Yaskawa INFORM job: SKRZYNIA_5540_-90_STOPNI_10BR.JBI

/JOB
//NAME SKRZYNIA_5540_-90_STOPNI_10BR
///FOLDERNAME 02-SKRZYNIE_JOBS
//POS
///NPOS 690,690,0,51,0,0
///TOOL 0
///POSTYPE PULSE
///PULSE
C00000=0,-52280,40443,0,6876,0
C00001=-82314,-24956,17040,-59626,-27382,-6248
C00002=-93910,-8625,17040,-59626,-43355,-6248
C00003=-98846,-1061,-42166,-80308,-57081,16120
C00004=-100452,6057,-48127,-85711,-56704,21322
C00005=-96957,25597,-37888,-85158,-62082,25522
C00006=-95580,33075,-33256,-84644,-64024,26851
C00007=-94380,33739,-32188,-85134,-63496,26721
C00008=-95580,33075,-33256,-84644,-64024,26851
C00009=-94940,31262,-36138,-85248,-63712,27160
C00010=-95580,33075,-33256,-84644,-64024,26851
C00011=-95263,33142,-33256,-84677,-63995,26850
C00012=-95263,33142,-33256,-84677,-63995,26850
C00013=-94261,33702,-32359,-85087,-63552,26740
C00014=-95263,33142,-33256,-84677,-63995,26850
C00015=-94777,31773,-35433,-85135,-63758,27084
C00016=-95263,33142,-33256,-84677,-63995,26850
C00017=-95260,33144,-33256,-84678,-63995,26850
C00018=-95260,33144,-33256,-84678,-63995,26850
C00019=-94282,33689,-32380,-85076,-63563,26742
C00020=-95260,33144,-33256,-84678,-63995,26850
C00021=-94827,31920,-35204,-85086,-63784,27059
C00022=-95260,33144,-33256,-84678,-63995,26850
C00023=-95258,33145,-33257,-84676,-63996,26846
C00024=-95258,33145,-33257,-84676,-63996,26846
C00025=-94286,33686,-32387,-85074,-63568,26738
C00026=-95258,33145,-33257,-84676,-63996,26846
C00027=-94874,32057,-34990,-85039,-63809,27032
C00028=-95258,33145,-33257,-84676,-63996,26846
C00029=-95258,33145,-33257,-84676,-63996,26846
C00030=-95258,33145,-33257,-84676,-63996,26846
C00031=-94323,33667,-32422,-85059,-63584,26741
C00032=-95258,33145,-33257,-84676,-63996,26846
C00033=-94899,32130,-34875,-85014,-63820,27019
C00034=-95258,33145,-33257,-84676,-63996,26846
C00035=-95258,25631,32269,-66559,-75499,2416
C00036=-95258,25631,32269,-66559,-75499,2416
C00037=-94333,26371,33350,-66433,-74983,2224
C00038=-95258,25631,32269,-66559,-75499,2416
C00039=-94886,24142,30119,-66602,-75133,2534
C00040=-95258,25631,32269,-66559,-75499,2416
C00041=-98646,19496,-17631,-99827,-80462,21224
C00042=-98811,21047,-15512,-99242,-81394,20987
C00043=-97886,21574,-14788,-99528,-80824,20997
C00044=-98811,21047,-15512,-99242,-81394,20987
C00045=-98517,19954,-17009,-99363,-81263,21101
C00046=-98811,21047,-15512,-99242,-81394,20987
C00047=-98811,19937,1242,-97498,-78933,15296
C00048=-98811,19937,1242,-97498,-78933,15296
C00049=-97933,20465,1962,-97646,-78345,15298
C00050=-98811,19937,1242,-97498,-78933,15296
C00051=-98523,18806,-285,-97586,-78782,15407
C00052=-98811,19937,1242,-97498,-78933,15296
C00053=-99152,37522,67957,-90787,-75030,-95
C00054=-99152,37522,67957,-90787,-75030,-95
C00055=-98279,38495,69612,-90504,-74443,-274
C00056=-99152,37522,67957,-90787,-75030,-95
C00057=-98708,34478,62881,-90983,-74820,488
C00058=-99152,37522,67957,-90787,-75030,-95
C00059=-98988,22776,44546,-90608,-68570,2568
C00060=-94428,854,16076,-89248,-50738,4740
C00061=-88080,-20128,-3199,-80943,-31244,2335
C00062=-50003,-39410,-5978,-16260,-18649,-25999
C00063=-48287,-44591,-17414,-16172,-14532,-25809
C00064=-91598,-4780,31748,-51735,-45731,-8771
C00065=-100979,4048,11685,-70926,-63965,7529
C00066=-99314,21122,10686,-75447,-74504,15845
C00067=-95042,27764,23446,-66422,-76166,12644
C00068=-94670,26279,21282,-66499,-75794,12766
C00069=-95042,27764,23446,-66422,-76166,12644
C00070=-94070,28550,24602,-66381,-75626,12438
C00071=-95042,27764,23446,-66422,-76166,12644
C00072=-97373,30352,38967,-71736,-79717,10385
C00073=-97373,30352,38967,-71736,-79717,10385
C00074=-96432,31128,40151,-71627,-79165,10198
C00075=-97373,30352,38967,-71736,-79717,10385
C00076=-97071,28917,36802,-71776,-79407,10544
C00077=-97373,30352,38967,-71736,-79717,10385
C00078=-97356,30262,38827,-71739,-79698,10398
C00079=-97356,30262,38827,-71739,-79698,10398
C00080=-96507,30957,39891,-71642,-79201,10230
C00081=-97356,30262,38827,-71739,-79698,10398
C00082=-97092,29010,36937,-71773,-79425,10538
C00083=-97356,30262,38827,-71739,-79698,10398
C00084=-97431,30641,39402,-71725,-79780,10352
C00085=-97431,30641,39402,-71725,-79780,10352
C00086=-96578,31348,40481,-71627,-79280,10181
C00087=-97431,30641,39402,-71725,-79780,10352
C00088=-97114,29116,37095,-71767,-79448,10523
C00089=-97431,30641,39402,-71725,-79780,10352
C00090=-99739,25677,21114,-82085,-78790,-4409
C00091=-99739,25677,21114,-82085,-78790,-4409
C00092=-98872,26250,21941,-82102,-78216,-4501
C00093=-99739,25677,21114,-82085,-78790,-4409
C00094=-99422,24232,19045,-82158,-78544,-4261
C00095=-99739,25677,21114,-82085,-78790,-4409
C00096=-98070,21699,18791,-100677,-76082,-5031
C00097=-98401,27942,27737,-100067,-79473,-6121
C00098=-97586,28537,28617,-100081,-78897,-6135
C00099=-98401,27942,27737,-100067,-79473,-6121
C00100=-98064,26400,25481,-100144,-79339,-5917
C00101=-98401,27942,27737,-100067,-79473,-6121
C00102=-99160,29228,35009,-99418,-79080,-8034
C00103=-98369,30564,38686,-99156,-78226,-8682
C00104=-97572,31199,39655,-99108,-77655,-8715
C00105=-98369,30564,38686,-99156,-78226,-8682
C00106=-98044,28949,36247,-99232,-78106,-8445
C00107=-98369,30564,38686,-99156,-78226,-8682
C00108=-99703,29561,37167,-99227,-79176,-8639
C00109=-98419,30528,38631,-99158,-78261,-8681
C00110=-98025,28599,35720,-99249,-78116,-8401
C00111=-98419,30528,38631,-99158,-78261,-8681
C00112=-97391,31350,39887,-99096,-77526,-8725
C00113=-98419,30528,38631,-99158,-78261,-8681
C00114=-91461,-8162,-10615,-106368,-48885,623
C00115=-98486,-14751,-40891,-114294,-59712,7739
C00116=-84089,-24462,-58822,-138905,-52068,17717
C00117=-93370,-29108,-64994,-133695,-56362,15444
C00118=-62749,-65297,-81682,-146767,-31843,20298
C00119=-73187,-23116,26488,-26118,-57509,-28469
C00120=-88600,6462,53521,-37454,-59134,-23478
C00121=-98388,13381,40686,-64111,-66922,-10378
C00122=-99819,33446,48735,-87787,-79679,-1235
C00123=-99819,33446,48735,-87787,-79679,-1235
C00124=-98945,34179,49898,-87659,-79086,-1350
C00125=-99819,33446,48735,-87787,-79679,-1235
C00126=-99591,32133,46677,-87830,-79529,-1033
C00127=-99819,33446,48735,-87787,-79679,-1235
C00128=-98853,28116,28355,-96898,-79749,4777
C00129=-98853,30464,37910,-96149,-78952,2546
C00130=-98284,30904,38579,-96116,-78548,2515
C00131=-98853,30464,37910,-96149,-78952,2546
C00132=-98656,29478,36421,-96191,-78865,2688
C00133=-98853,30464,37910,-96149,-78952,2546
C00134=-100018,29602,36606,-96210,-79777,2602
C00135=-100018,29602,36606,-96210,-79777,2602
C00136=-99324,30109,37370,-96174,-79287,2570
C00137=-99039,28675,35212,-96234,-79160,2773
C00138=-99324,30109,37370,-96174,-79287,2570
C00139=-98210,30963,38666,-96111,-78498,2511
C00140=-99324,30109,37370,-96174,-79287,2570
C00141=-94437,3365,15121,-90804,-55123,21
C00142=-76606,-19838,2636,-59027,-23020,-13375
C00143=-49667,-45532,-21960,-5654,-17518,-35856
C00144=-47485,-50287,-32535,-1070,-13732,-37871
///LIMIT ON
C00145=-36103,-65917,11738,-26975,4295,7905
///LIMIT OFF
C00146=-48283,-21883,28214,-25170,-26491,48363
C00147=-46664,-3144,58041,-18842,-32105,45325
C00148=-50347,-18571,12268,-49104,-16423,60029
C00149=-53571,-17125,12073,-56866,-17385,63433
C00150=-52069,-15730,13206,-55612,-16432,62999
C00151=-53474,-15384,13495,-57637,-17161,63825
C00152=-53571,-17125,12073,-56866,-17385,63433
C00153=-50509,-19000,10610,-51503,-15997,61182
C00154=-53130,-17211,12007,-56251,-17152,63186
C00155=-51822,-15992,12994,-55136,-16324,62798
C00156=-53635,-15431,13457,-57815,-17251,63894
C00157=-53130,-17211,12007,-56251,-17152,63186
C00158=-50704,-18403,11069,-52157,-16018,61478
C00159=-53231,-16470,14622,-53206,-17893,61673
C00160=-51756,-15101,15744,-51790,-16990,61165
C00161=-53741,-14453,16285,-54808,-17949,62397
C00162=-53231,-17580,11714,-56182,-17246,63139
C00163=-51814,-19410,10295,-53186,-16720,61844
C00164=-53629,-18979,7405,-62018,-16535,65958
C00165=-52238,-17698,8415,-61175,-15613,65699
C00166=-53551,-17401,8655,-62910,-16346,66402
C00167=-52880,-17654,11656,-55678,-17066,62935
C00168=-51005,-17995,11387,-52847,-16122,61778
C00169=-52964,-17611,11689,-55811,-17106,62990
C00170=-51611,-16353,12697,-54642,-16249,62582
C00171=-53495,-15765,13180,-57466,-17201,63739
C00172=-52964,-17611,11689,-55811,-17106,62990
C00173=-51030,-17982,11395,-52891,-16135,61798
C00174=-52975,-17563,11726,-55850,-17109,63009
C00175=-51607,-16289,12749,-54669,-16241,62596
C00176=-53283,-15811,13140,-57177,-17094,63622
C00177=-52975,-17563,11726,-55850,-17109,63009
C00178=-50945,-18019,11363,-52741,-16103,61737
C00179=-52728,-17788,11545,-55393,-17010,62816
C00180=-51045,-16207,12813,-53894,-15944,62287
C00181=-52895,-15647,13274,-56746,-16874,63461
C00182=-52728,-17788,11545,-55393,-17010,62816
C00183=-50945,-18019,11363,-52741,-16103,61737
C00184=-52556,-17520,11756,-55311,-16888,62798
C00185=-51113,-16157,12849,-54025,-15975,62343
C00186=-52730,-15718,13210,-56498,-16792,63358
C00187=-52556,-17520,11756,-55311,-16888,62798
C00188=-50945,-18019,11363,-52741,-16103,61737
C00189=-51893,-17787,11546,-54246,-16568,62356
C00190=-50379,-16341,12703,-52826,-15610,61849
C00191=-52406,-15704,13225,-56071,-16614,63190
C00192=-51893,-17787,11546,-54246,-16568,62356
C00193=-50028,-22953,-3957,-22347,-31919,54220
C00194=-50947,-22502,-3625,-23433,-32061,54736
C00195=-49421,-20951,-2455,-21951,-31329,54057
C00196=-51207,-20433,-2055,-24026,-31698,55041
C00197=-50529,-22709,-3778,-22940,-31995,54502
C00198=-49763,-25421,-36239,-24565,-26935,60445
C00199=-49763,-25421,-36239,-24565,-26935,60445
C00200=-48299,-23485,-34758,-23276,-26122,59713
C00201=-50218,-22723,-34165,-25568,-26529,60993
C00202=-49763,-25421,-36239,-24565,-26935,60445
C00203=-50713,-12366,-58367,-41124,-17813,74400
C00204=-50824,-12254,-58263,-41255,-17847,74484
C00205=-49431,-10052,-56192,-40383,-17131,73813
C00206=-50915,-9358,-55524,-41955,-17664,74847
C00207=-51028,-12852,-58814,-41301,-17980,74542
C00208=-49763,-25421,-36239,-24565,-26935,60445
C00209=-50529,-22709,-3778,-22940,-31995,54502
C00210=-45389,-28224,4312,-35967,-15579,54278
C00211=-40154,-51179,-915,-24203,-8234,36524
C00212=0,-52280,40443,0,6876,0
C00213=0,-52280,40443,0,6876,0
C00214=-2117,-50103,-33543,-4117,45077,85249
C00215=26439,-48928,-33543,-4117,-52362,85249
C00216=26439,-27355,-33543,-41485,-52362,85249
C00217=39218,-24492,-41653,-51934,-39374,86964
C00218=39218,-24492,-41653,-51934,-39374,86964
C00219=46639,7575,-9331,-26045,-41627,82486
C00220=47278,8641,-9483,-26175,-40625,82510
C00221=46369,10567,-7126,-26545,-41054,82831
C00222=47278,8641,-9483,-26175,-40625,82510
C00223=48256,9506,-8430,-25641,-40400,82076
C00224=47278,8641,-9483,-26175,-40625,82510
C00225=44522,-635,-31983,-49264,-28311,89687
C00226=44247,-628,-31975,-49394,-28443,89790
C00227=43310,1314,-29842,-49807,-28910,90140
C00228=44247,-628,-31975,-49394,-28443,89790
C00229=45313,152,-31124,-48894,-27920,89380
C00230=44247,-628,-31975,-49394,-28443,89790
C00231=41572,-13073,-22520,-50760,-38355,84033
C00232=21909,-6773,-14577,-94161,-56302,89381
C00233=23773,-3183,-10897,-94486,-55065,89563
C00234=24904,-823,-8382,-94654,-54308,89644
C00235=24395,1151,-6219,-94590,-54651,89617
C00236=24904,-823,-8382,-94654,-54308,89644
C00237=26178,-337,-7854,-94816,-53451,89710
C00238=24904,-823,-8382,-94654,-54308,89644
C00239=17020,-16061,-23281,-93084,-59494,88637
C00240=-21568,-26506,-31664,-90508,-85573,86639
C00241=-8557,-39769,-22319,-51419,-69406,84680
C00242=-8557,-39769,-22319,-51419,-69406,84680
C00243=32994,-9735,-10751,-29019,-59471,69498
C00244=43974,9628,-22604,-36190,-36396,73426
C00245=45932,13115,-22315,-37472,-33732,73846
C00246=45228,14664,-20329,-37571,-34159,74020
C00247=45932,13115,-22315,-37472,-33732,73846
C00248=46653,13731,-21526,-37109,-33514,73520
C00249=45932,13115,-22315,-37472,-33732,73846
C00250=39039,866,-6986,-42761,-44691,67687
C00251=30717,-9248,-22721,-77433,-42696,79486
C00252=32434,-7077,-20587,-77571,-41526,79457
C00253=31883,-5576,-19073,-77676,-41878,79560
C00254=32434,-7077,-20587,-77571,-41526,79457
C00255=33092,-6769,-20280,-77576,-41084,79417
C00256=32434,-7077,-20587,-77571,-41526,79457
C00257=30527,-14106,-27266,-76898,-42917,79150
C00258=25454,-9581,-17335,-94425,-53880,89429
C00259=24965,-2445,-10120,-94645,-54263,89631
C00260=24893,-1278,-8874,-94650,-54314,89639
C00261=24417,557,-6877,-94595,-54636,89618
C00262=24893,-1278,-8874,-94650,-54314,89639
C00263=25752,-956,-8526,-94759,-53737,89684
C00264=24893,-1278,-8874,-94650,-54314,89639
C00265=23817,-1527,-9142,-94518,-55040,89587
C00266=24871,-1152,-8735,-94651,-54328,89643
C00267=24440,508,-6926,-94601,-54619,89624
C00268=24871,-1152,-8735,-94651,-54328,89643
C00269=25635,-865,-8427,-94748,-53815,89684
C00270=24871,-1152,-8735,-94651,-54328,89643
C00271=33203,-4295,-13750,-123758,-49995,81034
C00272=35028,4195,-6818,-132965,-58836,87950
C00273=35028,4195,-6818,-132965,-58836,87950
C00274=34452,5837,-4911,-132720,-59045,87770
C00275=35028,4195,-6818,-132965,-58836,87950
C00276=35710,4593,-6360,-133217,-58512,88125
C00277=35028,4195,-6818,-132965,-58836,87950
C00278=24762,-11408,-28656,-113055,-60293,85383
C00279=-28645,-26349,-41223,-103369,-91870,78302
C00280=-28645,-26349,-41223,-103369,-91870,78302
C00281=-25549,-24286,-26215,-66769,-87032,80148
C00282=27561,-8271,-12315,-63268,-52553,74387
C00283=29336,-165,-3925,-63163,-51316,74265
C00284=29518,765,-2904,-63127,-51205,74233
C00285=28850,2962,-447,-63227,-51636,74327
C00286=29518,765,-2904,-63127,-51205,74233
C00287=30662,1292,-2320,-62902,-50501,74035
C00288=29518,765,-2904,-63127,-51205,74233
C00289=30773,10953,32136,-106912,-46141,83783
C00290=30773,10953,32136,-106912,-46141,83783
C00291=30080,13410,35293,-106601,-46463,83481
C00292=30773,10953,32136,-106912,-46141,83783
C00293=32007,11622,32987,-106899,-45346,83915
C00294=30773,10953,32136,-106912,-46141,83783
C00295=28321,-8642,-16372,-95739,-47180,89965
C00296=28583,-7344,-15096,-95864,-47019,90043
C00297=27897,-5229,-12965,-95873,-47499,90079
C00298=28583,-7344,-15096,-95864,-47019,90043
C00299=29900,-6813,-14567,-96101,-46141,90154
C00300=28583,-7344,-15096,-95864,-47019,90043
C00301=27852,-7537,-15286,-95742,-47508,89986
C00302=28448,-7306,-15058,-95845,-47110,90035
C00303=27795,-5283,-13021,-95851,-47567,90065
C00304=28448,-7306,-15058,-95845,-47110,90035
C00305=29772,-6774,-14527,-96083,-46226,90146
C00306=28448,-7306,-15058,-95845,-47110,90035
C00307=18552,-19531,-26179,-93438,-53589,88597
C00308=40301,-14999,-52277,-148979,-69262,86714
C00309=42323,-33,-37432,-150113,-69667,87489
C00310=53245,19091,3515,-165691,-72595,90030
C00311=53641,19552,4138,-165817,-72473,90151
C00312=53058,20743,5761,-165615,-72317,89948
C00313=53641,19552,4138,-165817,-72473,90151
C00314=54155,20160,4967,-165982,-72308,90306
C00315=53641,19552,4138,-165817,-72473,90151
C00316=23439,-10154,-17205,-109204,-58547,76547
C00317=2382,-21913,-40813,-107544,-74451,77239
C00318=-31257,-15877,-35733,-102288,-96107,74463
C00319=-39204,-18003,-7668,-86141,-99190,68413
C00320=-5592,-5690,18047,-75373,-79525,63129
C00321=19039,-439,25862,-68224,-64120,61443
C00322=21624,5223,26011,-69375,-61155,63193
C00323=24437,11840,34139,-68260,-59598,62567
C00324=24053,13588,36402,-68249,-59917,62491
C00325=24437,11840,34139,-68260,-59598,62567
C00326=25079,12112,34488,-68051,-59212,62472
C00327=24437,11840,34139,-68260,-59598,62567
C00328=21370,4935,25667,-69451,-61310,63230
C00329=-18351,-11002,3811,-80352,-86206,66275
C00330=-34619,-5846,8788,-82342,-97004,67025
C00331=-40684,-19963,-8478,-86482,-100204,67987
C00332=1570,-13136,-5998,-86227,-71173,69099
C00333=13966,-6596,-2340,-86587,-62612,70052
C00334=24093,-1862,-9504,-94546,-54850,89594
C00335=24093,-1862,-9504,-94546,-54850,89594
C00336=23519,425,-7024,-94488,-55240,89573
C00337=24093,-1862,-9504,-94546,-54850,89594
C00338=25256,-1442,-9053,-94693,-54067,89656
C00339=24093,-1862,-9504,-94546,-54850,89594
C00340=27718,4364,12871,-105518,-51077,86669
C00341=27718,4364,12871,-105518,-51077,86669
C00342=27164,6353,15202,-105385,-51398,86539
C00343=27718,4364,12871,-105518,-51077,86669
C00344=28828,4851,13441,-105618,-50355,86801
C00345=27718,4364,12871,-105518,-51077,86669
C00346=20930,-1364,27707,-95004,-52134,77785
C00347=-41463,-32191,18163,-91991,-64949,55938
C00348=0,-52277,40442,0,6872,4
C00349=-82314,-24956,17040,-59626,-27382,-6248
C00350=-93910,-8625,17040,-59626,-43355,-6248
C00351=-98846,-1061,-42166,-80308,-57081,16120
C00352=-100452,6057,-48127,-85711,-56704,21322
C00353=-95564,34698,-34234,-85516,-63941,27819
C00354=-94221,34299,-28769,-82558,-65564,25844
C00355=-94107,37241,-30442,-84005,-65307,27544
C00356=-95103,32620,-31323,-83378,-64939,26072
C00357=-95103,32620,-31323,-83378,-64939,26072
C00358=-93990,32828,-31380,-83932,-64473,26160
C00359=-94063,31710,-30585,-83283,-64598,25457
C00360=-96692,32939,-31211,-82617,-65723,26190
C00361=-96111,21840,170,-71736,-70232,11396
C00362=-94229,22391,773,-71789,-70557,11468
C00363=-94283,22521,1025,-71678,-70686,11433
C00364=-95675,19167,-4176,-72970,-68231,11735
C00365=-95681,24338,3488,-71459,-71669,11415
C00366=-94245,22750,1246,-71757,-70674,11453
C00367=-94341,22923,1499,-71729,-70746,11440
C00368=-96213,24222,3324,-71394,-71999,11479
C00369=-95517,23330,2066,-71543,-71508,11507
C00370=-94304,22892,1449,-71738,-70721,11443
C00371=-94158,22889,1452,-71756,-70627,11429
C00372=-96071,24319,3461,-71408,-71916,11455
C00373=-96941,-6406,-33809,-76117,-54125,10511
C00374=-89093,-33107,-44597,-67545,-52550,2722
C00375=-66103,-61757,7450,-21008,-32955,-5749
C00376=4223,-52290,40457,-5766,6913,3980
C00377=4223,-52290,40457,-5766,6913,3980
C00378=-4538,-50065,-33535,-3011,44998,84219
C00379=24207,-49248,-33668,-5551,-52644,86091
C00380=25094,-27722,-33812,-41887,-53054,85599
C00381=38036,-25052,-42086,-52219,-40087,87228
C00382=37328,-2824,-24733,-57182,-37821,90318
C00383=36700,-2520,-13735,-51589,-42201,86442
C00384=37520,2330,-3498,-48550,-43875,84431
C00385=37520,1020,-12079,-52650,-40851,87066
C00386=48458,-261,-12985,-24069,-43340,80504
C00387=36153,7296,-1758,-40139,-50302,89334
C00388=37146,11264,2520,-40849,-50296,89553
C00389=38059,11410,-1863,-40565,-47910,90206
C00390=36726,6476,-7858,-41213,-48206,90783
C00391=19339,7883,9818,-77509,-64249,74140
C00392=19027,1888,-16187,-103553,-67480,82955
C00393=24158,3537,-14322,-106039,-60939,84018
C00394=24143,4321,-7309,-103852,-59670,81875
C00395=19531,2904,-8928,-102027,-65985,80961
C00396=20232,-3383,-14682,-86495,-63009,78978
C00397=-24375,-51634,-49601,-83793,-94064,73950
C00398=4223,-52290,40457,-5766,6913,3980
C00399=-4825,-36686,24602,37792,-30278,35378
C00400=-46221,-29633,7403,-27051,-24124,46751
C00401=-46221,-29633,7403,-27051,-24124,46751
C00402=-52474,-20611,11454,-41004,-23045,52959
C00403=-60257,-19980,-2088,-84190,-23320,82051
C00404=-63868,-19883,-6318,-95759,-28031,88346
C00405=-51819,-22965,8574,-41365,-22900,53139
C00406=-4825,-36686,24602,37792,-30278,35378
C00407=-66103,-61757,7450,-21008,-32955,-5749
C00408=-89093,-33107,-44597,-67545,-52550,2722
C00409=-96941,-6406,-33809,-76117,-54125,10511
C00410=-99429,14378,84,-80785,-71596,8628
C00411=-99699,24313,24829,-82602,-77917,4569
C00412=-98066,26841,20697,-83331,-79245,6860
C00413=-98079,26929,20513,-83349,-79351,6953
C00414=-99638,19663,10292,-84193,-74452,7551
C00415=-99636,19665,10291,-84197,-74448,7550
C00416=-98131,26698,20177,-83371,-79212,6975
C00417=-98097,25980,12653,-84102,-79057,9159
C00418=-99636,19665,10291,-84197,-74448,7550
C00419=-99636,19665,10291,-84197,-74448,7550
C00420=-98186,26934,20517,-83350,-79332,6954
C00421=-98240,27087,20738,-83333,-79465,6940
C00422=-99636,19665,10291,-84197,-74448,7550
C00423=-99215,3992,8526,-80547,-63068,1835
C00424=-100264,1107,23397,-72827,-59854,-5092
C00425=-100264,1107,23397,-72827,-59854,-5092
C00426=-99514,-9483,18258,-71284,-60958,-4118
C00427=-61441,-38616,11032,-55510,-42874,-3049
C00428=4223,-52290,40457,-5766,6913,3980
C00429=-22331,-23394,-30093,-82917,-82006,85712
C00430=22434,-14401,-3235,-51104,-60845,74728
C00431=42744,21307,45077,-24753,-69813,65333
C00432=33655,14083,18147,-45417,-58301,71861
C00433=33641,11943,8279,-47835,-54840,73983
C00434=36574,13250,23432,-35354,-61822,69159
C00435=28497,326,20939,-70981,-47632,72427
C00436=30972,5983,29862,-68494,-46670,70994
C00437=31029,11571,45127,-63398,-49004,67378
C00438=28971,8096,39948,-65070,-49810,68216
C00439=29759,-12862,-24221,-91747,-41905,86600
C00440=35278,-10419,-21940,-93284,-36771,87139
C00441=36208,-10883,-22374,-93618,-35345,87231
C00442=27219,-23595,-33313,-89555,-43517,85303
C00443=10564,-40773,-45889,-85382,-54876,82708
C00444=-14984,-61618,-24572,-87392,-53367,60735
C00445=9346,-67436,-18786,-75708,-34590,53709
C00446=40938,-55232,35946,-9746,5421,6718
C00447=4223,-52290,40457,-5766,6913,3980
C00448=-4825,-36686,24602,37792,-30278,35378
C00449=-46221,-29633,7403,-27051,-24124,46751
C00450=-56796,-22932,368,-68953,-21567,70907
C00451=-61611,-20349,-6598,-95791,-25091,88405
C00452=-63740,-19715,-7390,-98604,-28245,90373
C00453=-52085,-22687,8760,-40927,-22666,52970
C00454=-49294,-34086,9663,-30689,-30758,52546
C00455=4223,-52290,40457,-5766,6913,3980
C00456=0,-52280,40443,0,6876,0
C00457=0,-52280,40443,0,6876,0
C00458=-61754,-61602,7279,-16215,-32140,-7126
C00459=-89313,-24027,20291,-53466,-58905,-4975
C00460=-97807,-25409,-21837,-78881,-62828,2121
C00461=-95644,-21015,-18476,-76474,-46020,1039
C00462=-99784,20282,11129,-84157,-74554,7499
C00463=-100058,25789,39872,-88643,-74345,1113
C00464=-98402,30585,40634,-89771,-78826,2411
C00465=-98157,28480,31016,-94616,-79375,5454
C00466=-99711,20530,18234,-96341,-74733,7105
C00467=-98387,24449,13333,-103557,-81562,10447
C00468=-96604,24297,13119,-103804,-80422,10626
C00469=-96604,26005,23528,-102938,-78741,7977
C00470=-99312,16704,-2418,-105415,-78692,13344
C00471=-99082,-15666,-17237,-92076,-50940,5911
C00472=-62624,-50447,-44776,-76934,-16957,-1114
C00473=-75165,-16680,32803,-38944,-52307,-27215
C00474=-75165,-16680,32803,-38944,-52307,-27215
C00475=-95350,8536,58133,-52477,-59539,-22352
C00476=-100948,11380,23586,-76731,-68346,-5781
C00477=-95677,27971,29253,-68711,-77159,-3356
C00478=-95583,25946,19380,-69779,-75412,-992
C00479=-98294,19288,21509,-68095,-73058,-4657
C00480=-100497,3428,15340,-68921,-63273,-8271
C00481=-81087,-35886,-14825,-53529,-36311,-18004
C00482=-47029,-49867,-20464,-11808,-29290,-36568
///LIMIT ON
C00483=-41431,-67449,10869,-1325,127,-6150
///LIMIT OFF
C00484=6328,-52297,40483,-8599,6957,5944
C00485=-8648,-69005,-18270,-84275,-43232,53472
C00486=18757,-59462,-34892,-84638,-37529,67311
C00487=26772,-23733,-33422,-89486,-43820,85275
C00488=29039,-10071,-21608,-91386,-45181,86629
C00489=29639,-5923,-17523,-91591,-45648,86808
C00490=29709,-5453,-17046,-91618,-45636,86826
C00491=29138,-10182,-21714,-91372,-45196,86624
C00492=20424,-22725,-32635,-88800,-51006,85261
C00493=28416,-11420,-25238,-98178,-46636,84572
C00494=30481,-6584,-16425,-92636,-44382,82541
C00495=30464,-7521,-23523,-96665,-44944,85234
C00496=28416,-11420,-25238,-98178,-46636,84572
C00497=-23524,-33387,-42654,-89891,-81168,80229
C00498=-23524,-33387,-42654,-89891,-81168,80229
C00499=33935,-6399,-10013,-60506,-43064,77980
C00500=34878,-3211,-6740,-60356,-42422,77865
C00501=34873,-3218,-6748,-60357,-42424,77868
C00502=33935,-6399,-10013,-60506,-43064,77980
C00503=17782,-19597,1250,-60925,-51448,69151
C00504=-243,-43047,-13224,-69794,-55957,65877
C00505=42700,-55269,36176,-13619,5333,9062
C00506=6328,-52297,40483,-8599,6957,5944
C00507=-10231,-60460,6271,71658,-11927,-13637
C00508=-49129,-39322,3023,-34904,-18609,43900
C00509=-57258,-19535,13114,-46502,-25798,55150
C00510=-58736,-19151,1344,-78268,-22199,76919
C00511=-56868,-17231,8572,-62431,-21728,66645
C00512=-56011,-29317,6725,-41009,-27363,52457
C00513=-10137,-60963,4526,62308,-14518,-6745
C00514=0,-52280,40443,0,6876,0
C00515=0,-52280,40443,0,6876,0
C00516=-41653,-63035,2931,-3578,-7576,-14589
C00517=-45770,-50109,-20524,-10089,-29273,-37310
C00518=-80544,-36303,-15042,-52975,-36116,-18265
C00519=-98926,-23964,-13239,-67549,-54178,-9552
C00520=-98901,-11554,-2908,-69008,-53412,-8360
C00521=-101174,454,-4800,-81790,-63681,-152
C00522=-100336,15373,10036,-81991,-73209,850
C00523=-98655,27908,24922,-81730,-79774,792
C00524=-98593,28720,26118,-81685,-80145,709
C00525=-99951,24070,19376,-82000,-77829,1145
C00526=-99951,24070,19376,-82000,-77829,1145
C00527=-98577,27118,23759,-81796,-79157,859
C00528=-98518,28577,26461,-81649,-79882,537
C00529=-99951,24070,19376,-82000,-77829,1145
C00530=-99951,24070,19376,-82000,-77829,1145
C00531=-98479,26563,22955,-81844,-78651,906
C00532=-98651,28095,26058,-81646,-79654,489
C00533=-99951,24070,19376,-82000,-77829,1145
C00534=-97595,-1409,-12320,-84284,-60474,1798
C00535=-100010,-16422,-27011,-84227,-53565,945
C00536=-88098,-29848,-22776,-71580,-48483,-7812
C00537=-81694,-37220,-20464,-64791,-45723,-12569
C00538=-45770,-50109,-20524,-10089,-29273,-37310
///LIMIT ON
C00539=-40984,-65135,6743,-2520,-4051,-10897
///LIMIT OFF
C00540=0,-52280,40443,0,6876,0
C00541=40939,-55232,35946,-9746,5421,6719
C00542=8707,-69002,-18268,-75213,-34271,52581
C00543=23267,-58917,-25142,-81990,-31707,62852
C00544=27307,-5613,10331,-81857,-46454,76095
C00545=30064,-5598,-963,-91827,-44222,81590
C00546=30419,-1725,5291,-88668,-43977,80354
C00547=30554,-300,10432,-88528,-43656,79164
C00548=29815,-6351,-3652,-90193,-44535,81892
C00549=29567,1847,27834,-65726,-48411,69959
C00550=23257,11670,30420,-81328,-57342,77033
C00551=23257,16856,45442,-77525,-58254,73578
C00552=21577,7912,33836,-78698,-59121,74340
C00553=17856,-9033,24892,-70658,-55966,67475
C00554=20838,-7097,2019,-111788,-62648,79114
C00555=40635,280,-7982,-142398,-56681,90238
C00556=32653,-9455,434,-90251,-40347,77213
C00557=40635,572,-6271,-142064,-55879,89947
C00558=40665,7761,2001,-141975,-55632,89869
C00559=40707,9678,10648,-140211,-51894,88431
C00560=39416,1907,3178,-139370,-51839,87774
C00561=7767,-21333,-19174,-120411,-69473,77116
C00562=33666,-18553,20064,-54519,-41956,59729
C00563=4032,-43511,13506,-33366,-30942,40837
C00564=22997,-56875,21315,16958,-8102,3163
C00565=0,-52280,40443,0,6876,0
///LIMIT ON
C00566=-50974,-46557,23391,-77768,-13896,42026
///LIMIT OFF
C00567=-53474,-39983,4253,-39182,-18848,44272
C00568=-56619,-19856,12878,-45665,-25558,54806
C00569=-53298,-26712,-11188,-26889,-32979,52528
C00570=-57200,-20845,-7559,-37425,-33513,53351
C00571=-58648,-23818,-25853,-45100,-31207,62168
C00572=-58477,-22145,-38977,-48305,-29254,64725
C00573=-51868,-27423,-11673,-25269,-32728,51737
C00574=-49121,-45409,-2608,-26656,-19965,38583
C00575=-21301,-61008,4568,43957,-10534,-712
C00576=0,-52280,40443,0,6876,0
C00577=0,-52280,40443,0,6876,0
///LIMIT ON
C00578=-40221,-67507,11044,-1325,-65,-6716
///LIMIT OFF
C00579=-45770,-50109,-20525,-10088,-29274,-37311
C00580=-80544,-36303,-15042,-52975,-36116,-18265
C00581=-97467,-10562,-5788,-76786,-47590,-5366
C00582=-98581,16268,9073,-102291,-74115,5399
C00583=-96245,23653,15791,-106069,-78604,6508
C00584=-96042,26225,19489,-105739,-79656,6032
C00585=-98519,17635,7561,-106659,-77043,7343
C00586=-98519,17635,7561,-106659,-77043,7343
C00587=-96298,25666,18652,-105800,-79560,6117
C00588=-95268,26547,15396,-109206,-81354,7908
C00589=-98519,17635,7561,-106659,-77043,7343
C00590=-98519,17635,7561,-106659,-77043,7343
C00591=-96096,27437,22144,-104884,-80110,5412
C00592=-96096,29559,32298,-104067,-78465,2996
C00593=-99245,17823,12181,-105373,-75632,5896
C00594=-101192,5225,-3909,-107580,-71003,7673
C00595=-100287,-3253,-24038,-111364,-68562,12025
C00596=-99412,-19117,-26908,-100833,-57247,5735
C00597=-91712,-30589,-22890,-72058,-50969,-7685
C00598=-81694,-37221,-20464,-64791,-45723,-12569
C00599=-45770,-50109,-20525,-10088,-29274,-37311
///LIMIT ON
C00600=-40221,-67507,11044,-1325,-65,-6716
///LIMIT OFF
C00601=0,-52280,40443,0,6876,0
C00602=51241,-30653,28678,4016,-29070,6398
C00603=46185,-61941,-37286,-12736,-10732,51851
C00604=-13205,-44768,-23966,-65315,-59418,73750
C00605=-11120,-40541,-20876,-69249,-61539,75403
C00606=-836,-13033,12361,-83908,-73576,73378
C00607=18912,6214,32354,-79489,-60743,73080
C00608=21217,10898,38129,-78632,-59343,72736
C00609=23447,16313,45262,-77527,-58074,72177
C00610=23610,23756,64158,-73325,-59549,68283
C00611=18912,6214,32354,-79489,-60743,73080
C00612=-836,-13033,12361,-83908,-73576,73378
C00613=-20209,-39682,-20467,-71924,-67122,76479
C00614=-20209,-39682,-20467,-71924,-67122,76479
C00615=26353,-3691,11741,-61723,-54035,71160
C00616=29598,-2090,11073,-69087,-47235,76987
C00617=30217,-1844,4641,-75777,-45517,79979
C00618=29529,1742,11379,-68166,-49318,73572
C00619=24010,-9039,-4437,-79986,-50972,77255
C00620=24652,-10740,-12845,-99298,-50700,81949
C00621=28976,-2672,-4778,-100308,-47937,82653
C00622=31030,-2921,-9996,-112394,-49006,86348
C00623=24652,-10740,-12845,-99298,-50700,81949
C00624=-25637,-26222,-38592,-96633,-85474,81576
C00625=-36771,-16470,-4689,-95304,-89579,74076
C00626=-33704,-12343,7746,-85568,-87064,70052
C00627=4032,-43511,13506,-33366,-30942,40837
C00628=27500,-60047,23168,28912,-2679,-5784
C00629=0,-52280,40443,0,6876,0
///LIMIT ON
C00630=-50971,-46557,23390,-77766,-13895,42026
///LIMIT OFF
C00631=-53475,-39984,4253,-39182,-18848,44273
C00632=-56619,-19856,12878,-45665,-25558,54806
C00633=-57643,-27958,-8553,-51854,-24771,59787
C00634=-66195,-24410,-19095,-90567,-31132,85904
C00635=-63290,-24193,-14362,-80030,-27547,78073
C00636=-39040,-40975,-15408,-18643,-21575,44866
C00637=-11647,-69843,-10959,56399,-11165,-4616
C00638=-15394,-57237,30542,-10392,5525,8219
C00639=0,-52280,40443,0,6876,0
C00640=0,-52280,40443,0,6876,0
///LIMIT ON
C00641=-40221,-67507,11044,-1325,-65,-6716
///LIMIT OFF
C00642=-45770,-50109,-20525,-10088,-29274,-37311
C00643=-94648,-18162,1575,-63292,-43035,-13570
C00644=-99112,3606,8889,-81344,-61742,-3619
C00645=-98572,26113,23382,-85571,-78492,509
C00646=-98656,28006,28806,-88976,-79248,97
C00647=-99839,24479,25828,-85077,-77001,-891
C00648=-99133,24879,24637,-94741,-77121,-2989
C00649=-98191,27052,27787,-94567,-78528,-3332
C00650=-98227,29022,36334,-93788,-77894,-5388
C00651=-100426,22466,21877,-95586,-77332,-2808
C00652=-99354,26201,32225,-100574,-76808,-3840
C00653=-96710,26250,34212,-100282,-74747,-4257
C00654=-96874,35880,54576,-99674,-76365,-9625
C00655=-99006,18159,13355,-102982,-74997,-2069
C00656=-97772,10218,8448,-107701,-67594,4685
C00657=-93425,-10069,4368,-74507,-47150,-8636
C00658=-96059,-18596,-7139,-76413,-48563,-7500
C00659=-96347,-8336,27647,-69083,-51241,-16001
C00660=-70313,-35289,-4922,-51188,-38634,-20596
C00661=-81694,-37221,-20464,-64791,-45723,-12569
C00662=-45770,-50109,-20525,-10088,-29274,-37311
C00663=-41628,-63095,3038,-3547,-7472,-14475
C00664=4223,-52290,40457,-5766,6913,3980
C00665=4224,-52288,40457,-5773,6909,3978
C00666=4224,-52288,40457,-28770,-64753,45638
C00667=6548,2882,44080,-77825,-67624,70557
C00668=22702,21750,69443,-66118,-61597,67582
C00669=25585,21999,63350,-62249,-61285,68688
C00670=25777,17209,50811,-62979,-59886,70957
C00671=23226,22825,71113,-65575,-61542,67353
C00672=24931,14697,51677,-80718,-51653,72069
C00673=24746,14409,39758,-87518,-53542,76879
C00674=24784,21556,58944,-82031,-53873,72431
C00675=22657,12722,42993,-85587,-54940,74916
C00676=-4427,-20395,-7318,-104668,-69521,79317
C00677=768,-20151,-3587,-97758,-65802,76626
C00678=-14736,-21545,-1233,-93598,-60476,72578
C00679=1642,-46684,14475,-47609,-24983,34912
C00680=27500,-60047,23168,28912,-2679,-5784
C00681=0,-52280,40443,0,6876,0
///LIMIT ON
C00682=-50971,-46557,23390,-77766,-13895,42026
///LIMIT OFF
C00683=-53475,-39984,4253,-39182,-18848,44273
C00684=-56619,-19856,12878,-45665,-25558,54806
C00685=-53891,-17708,14512,-43170,-23995,53902
C00686=-60674,-17500,6427,-71116,-24772,71097
C00687=-63181,-17997,2063,-82122,-26831,78394
C00688=-39402,-27697,7664,-17904,-21663,43170
C00689=-11647,-69843,-10959,56399,-11165,-4616
BC00000=479725
BC00001=460491
BC00002=460491
BC00003=460491
BC00004=460491
BC00005=460491
BC00006=460491
BC00007=460491
BC00008=460491
BC00009=460491
BC00010=460491
BC00011=506593
BC00012=506593
BC00013=506593
BC00014=506593
BC00015=506593
BC00016=506593
BC00017=552803
BC00018=552803
BC00019=552803
BC00020=552803
BC00021=552803
BC00022=552803
BC00023=598907
BC00024=598907
BC00025=598907
BC00026=598907
BC00027=598907
BC00028=598907
BC00029=621955
BC00030=621955
BC00031=621955
BC00032=621955
BC00033=621955
BC00034=621955
BC00035=574754
BC00036=574754
BC00037=574754
BC00038=574754
BC00039=574754
BC00040=574754
BC00041=620864
BC00042=620864
BC00043=620865
BC00044=620864
BC00045=620864
BC00046=620864
BC00047=620864
BC00048=620864
BC00049=620864
BC00050=620864
BC00051=620864
BC00052=620864
BC00053=619616
BC00054=619616
BC00055=619616
BC00056=619616
BC00057=619616
BC00058=619616
BC00059=619616
BC00060=619616
BC00061=619616
BC00062=619616
BC00063=714482
BC00064=722304
BC00065=754708
BC00066=767117
BC00067=767117
BC00068=767117
BC00069=767117
BC00070=767117
BC00071=767117
BC00072=752564
BC00073=752564
BC00074=752564
BC00075=752564
BC00076=752564
BC00077=752564
BC00078=798636
BC00079=798636
BC00080=798636
BC00081=798636
BC00082=798636
BC00083=798636
BC00084=821725
BC00085=821725
BC00086=821725
BC00087=821725
BC00088=821725
BC00089=821725
BC00090=858551
BC00091=858551
BC00092=858551
BC00093=858551
BC00094=858551
BC00095=858551
BC00096=864565
BC00097=864565
BC00098=864565
BC00099=864565
BC00100=864565
BC00101=864565
BC00102=879162
BC00103=879162
BC00104=879162
BC00105=879162
BC00106=879162
BC00107=879162
BC00108=916154
BC00109=916154
BC00110=916154
BC00111=916154
BC00112=916154
BC00113=916154
BC00114=887605
BC00115=887605
BC00116=887605
BC00117=887605
BC00118=887605
BC00119=974304
BC00120=974304
BC00121=984323
BC00122=988419
BC00123=988419
BC00124=988419
BC00125=988419
BC00126=988419
BC00127=988419
BC00128=1003836
BC00129=1003836
BC00130=1003836
BC00131=1003836
BC00132=1003836
BC00133=1003836
BC00134=1003836
BC00135=1048824
BC00136=1048824
BC00137=1048824
BC00138=1048824
BC00139=1048824
BC00140=1048824
BC00141=992185
BC00142=986127
BC00143=1002338
BC00144=951360
BC00145=873120
BC00146=935062
BC00147=935062
BC00148=964364
BC00149=966461
BC00150=966461
BC00151=966461
BC00152=966461
BC00153=904985
BC00154=904985
BC00155=904985
BC00156=904985
BC00157=904985
BC00158=843543
BC00159=843543
BC00160=843543
BC00161=843543
BC00162=843543
BC00163=782113
BC00164=782113
BC00165=782113
BC00166=782113
BC00167=782113
BC00168=720711
BC00169=720711
BC00170=720711
BC00171=720711
BC00172=720711
BC00173=659226
BC00174=659226
BC00175=659226
BC00176=659226
BC00177=659226
BC00178=597825
BC00179=597825
BC00180=597825
BC00181=597825
BC00182=597825
BC00183=536353
BC00184=536353
BC00185=536353
BC00186=536353
BC00187=536353
BC00188=474901
BC00189=474901
BC00190=474901
BC00191=474901
BC00192=474901
BC00193=474905
BC00194=474905
BC00195=474905
BC00196=474905
BC00197=474905
BC00198=474905
BC00199=474905
BC00200=474905
BC00201=474905
BC00202=474905
BC00203=474905
BC00204=474905
BC00205=474905
BC00206=474905
BC00207=474905
BC00208=474905
BC00209=474905
BC00210=474901
BC00211=548577
BC00212=548577
BC00213=492150
BC00214=423885
BC00215=423885
BC00216=423885
BC00217=423885
BC00218=423885
BC00219=493160
BC00220=493160
BC00221=493160
BC00222=493160
BC00223=493160
BC00224=493160
BC00225=539180
BC00226=539180
BC00227=539180
BC00228=539180
BC00229=539180
BC00230=539180
BC00231=525487
BC00232=485388
BC00233=485386
BC00234=485384
BC00235=485384
BC00236=485384
BC00237=485384
BC00238=485384
BC00239=485384
BC00240=485384
BC00241=485384
BC00242=635507
BC00243=635507
BC00244=635507
BC00245=635509
BC00246=635509
BC00247=635509
BC00248=635509
BC00249=635509
BC00250=603035
BC00251=594948
BC00252=594948
BC00253=594948
BC00254=594948
BC00255=594948
BC00256=594948
BC00257=594948
BC00258=600591
BC00259=600589
BC00260=600589
BC00261=600589
BC00262=600589
BC00263=600589
BC00264=600589
BC00265=623637
BC00266=623637
BC00267=623637
BC00268=623637
BC00269=623637
BC00270=623637
BC00271=623637
BC00272=623637
BC00273=623637
BC00274=623637
BC00275=623637
BC00276=623637
BC00277=623637
BC00278=623637
BC00279=623637
BC00280=758391
BC00281=758391
BC00282=758391
BC00283=758391
BC00284=758391
BC00285=758391
BC00286=758391
BC00287=758391
BC00288=758391
BC00289=669704
BC00290=669704
BC00291=669706
BC00292=669704
BC00293=669704
BC00294=669704
BC00295=784942
BC00296=784942
BC00297=784942
BC00298=784942
BC00299=784942
BC00300=784942
BC00301=807985
BC00302=807985
BC00303=807985
BC00304=807985
BC00305=807985
BC00306=807985
BC00307=807985
BC00308=784942
BC00309=784942
BC00310=784942
BC00311=784942
BC00312=784942
BC00313=784942
BC00314=784942
BC00315=784942
BC00316=785203
BC00317=785203
BC00318=785203
BC00319=895226
BC00320=895226
BC00321=895226
BC00322=895226
BC00323=895226
BC00324=895226
BC00325=895226
BC00326=895226
BC00327=895226
BC00328=895226
BC00329=906894
BC00330=906894
BC00331=963281
BC00332=963281
BC00333=963281
BC00334=969297
BC00335=969297
BC00336=969297
BC00337=969297
BC00338=969297
BC00339=969297
BC00340=969297
BC00341=969297
BC00342=969297
BC00343=969297
BC00344=969297
BC00345=969297
BC00346=927243
BC00347=899005
BC00348=490510
BC00349=460491
BC00350=460491
BC00351=460491
BC00352=460491
BC00353=460491
BC00354=461071
BC00355=460487
BC00356=461083
BC00357=499491
BC00358=507538
BC00359=497127
BC00360=507634
BC00361=488608
BC00362=495924
BC00363=488608
BC00364=496345
BC00365=534699
BC00366=542404
BC00367=534696
BC00368=534696
BC00369=565440
BC00370=565440
BC00371=557764
BC00372=557568
BC00373=557568
BC00374=557568
BC00375=557568
BC00376=557568
BC00377=492150
BC00378=423885
BC00379=471005
BC00380=487965
BC00381=477405
BC00382=472948
BC00383=455020
BC00384=453643
BC00385=453643
BC00386=493160
BC00387=521199
BC00388=521199
BC00389=521199
BC00390=521199
BC00391=484684
BC00392=484684
BC00393=484684
BC00394=484684
BC00395=484684
BC00396=484684
BC00397=484684
BC00398=508521
BC00399=598171
BC00400=670543
BC00401=670543
BC00402=670543
BC00403=670543
BC00404=731689
BC00405=732003
BC00406=598171
BC00407=557568
BC00408=557568
BC00409=606305
BC00410=572500
BC00411=559125
BC00412=566584
BC00413=559223
BC00414=566815
BC00415=605185
BC00416=605241
BC00417=605243
BC00418=605185
BC00419=628234
BC00420=635904
BC00421=628375
BC00422=628234
BC00423=628234
BC00424=599778
BC00425=599778
BC00426=599778
BC00427=599778
BC00428=599778
BC00429=590475
BC00430=610524
BC00431=594969
BC00432=594969
BC00433=594969
BC00434=593583
BC00435=552811
BC00436=552811
BC00437=552811
BC00438=552811
BC00439=612529
BC00440=612529
BC00441=620193
BC00442=620193
BC00443=620193
BC00444=620193
BC00445=620193
BC00446=620193
BC00447=635554
BC00448=828164
BC00449=903144
BC00450=912635
BC00451=916117
BC00452=977391
BC00453=977748
BC00454=868420
BC00455=557568
BC00456=557568
BC00457=557568
BC00458=557568
BC00459=589582
BC00460=608626
BC00461=608626
BC00462=628234
BC00463=633384
BC00464=640752
BC00465=648460
BC00466=648500
BC00467=692404
BC00468=692404
BC00469=692404
BC00470=692404
BC00471=648520
BC00472=648520
BC00473=665508
BC00474=721410
BC00475=729181
BC00476=752745
BC00477=779383
BC00478=779383
BC00479=779383
BC00480=766251
BC00481=748464
BC00482=748464
BC00483=748464
BC00484=748464
BC00485=620193
BC00486=626283
BC00487=635598
BC00488=635765
BC00489=635816
BC00490=643271
BC00491=641590
BC00492=641590
BC00493=685792
BC00494=685797
BC00495=685792
BC00496=685792
BC00497=685792
BC00498=771083
BC00499=750783
BC00500=758455
BC00501=750783
BC00502=750783
BC00503=719658
BC00504=685920
BC00505=620193
BC00506=635554
BC00507=576903
BC00508=514129
BC00509=423257
BC00510=423253
BC00511=484408
BC00512=484758
BC00513=539526
BC00514=539526
BC00515=748464
BC00516=748464
BC00517=748464
BC00518=748464
BC00519=763291
BC00520=763291
BC00521=783178
BC00522=785242
BC00523=786785
BC00524=794540
BC00525=786785
BC00526=809865
BC00527=809865
BC00528=816579
BC00529=809865
BC00530=855959
BC00531=855959
BC00532=862335
BC00533=855959
BC00534=855959
BC00535=855959
BC00536=855959
BC00537=855959
BC00538=810658
BC00539=756943
BC00540=748463
BC00541=620193
BC00542=700154
BC00543=704277
BC00544=716233
BC00545=716233
BC00546=716233
BC00547=716233
BC00548=716233
BC00549=733710
BC00550=733710
BC00551=733710
BC00552=733710
BC00553=742336
BC00554=742336
BC00555=742336
BC00556=763798
BC00557=742336
BC00558=742336
BC00559=742336
BC00560=742336
BC00561=743633
BC00562=750104
BC00563=672725
BC00564=672725
BC00565=688086
BC00566=591438
BC00567=480519
BC00568=423257
BC00569=423257
BC00570=423257
BC00571=423257
BC00572=423257
BC00573=423257
BC00574=486807
BC00575=539526
BC00576=539526
BC00577=748464
BC00578=748464
BC00579=748464
BC00580=768844
BC00581=788137
BC00582=849311
BC00583=861381
BC00584=868628
BC00585=861381
BC00586=884405
BC00587=884407
BC00588=891600
BC00589=884405
BC00590=915212
BC00591=915212
BC00592=915212
BC00593=915212
BC00594=885887
BC00595=883990
BC00596=875508
BC00597=855959
BC00598=855959
BC00599=810658
BC00600=748464
BC00601=748464
BC00602=762701
BC00603=816902
BC00604=816902
BC00605=837114
BC00606=816902
BC00607=816839
BC00608=816869
BC00609=816900
BC00610=816902
BC00611=816839
BC00612=816902
BC00613=837114
BC00614=903552
BC00615=903552
BC00616=897057
BC00617=903398
BC00618=903552
BC00619=903552
BC00620=903552
BC00621=903552
BC00622=903552
BC00623=903552
BC00624=903552
BC00625=848113
BC00626=815298
BC00627=672725
BC00628=672725
BC00629=688086
BC00630=591438
BC00631=529042
BC00632=550218
BC00633=573331
BC00634=572813
BC00635=633670
BC00636=633763
BC00637=633763
BC00638=633763
BC00639=633763
BC00640=748464
BC00641=748464
BC00642=991111
BC00643=983968
BC00644=997835
BC00645=1008455
BC00646=1005475
BC00647=1002598
BC00648=1007899
BC00649=1007899
BC00650=1007899
BC00651=1007899
BC00652=1057125
BC00653=1057125
BC00654=1057125
BC00655=1057125
BC00656=1008455
BC00657=998009
BC00658=1008455
BC00659=968816
BC00660=952198
BC00661=855959
BC00662=810658
BC00663=764236
BC00664=748464
BC00665=852584
BC00666=921533
BC00667=921533
BC00668=923427
BC00669=923499
BC00670=923499
BC00671=923501
BC00672=932594
BC00673=943380
BC00674=943380
BC00675=943380
BC00676=963295
BC00677=934184
BC00678=929661
BC00679=754884
BC00680=672725
BC00681=672725
BC00682=765203
BC00683=772042
BC00684=792000
BC00685=792000
BC00686=792000
BC00687=853734
BC00688=853356
BC00689=812121
///POSTYPE BASE
///RECTAN
///RCONF 1,0,0,0,0,0,0,0,0,0,0,0,0,0,0,0,0,0,0,0,0,0,0,0
P00006=0.000,0.000,0.000,0.0000,0.0000,0.0000
///RCONF 0,0,0,0,0,0,0,0,0,0,0,0,0,0,0,0,0,0,0,0,0,0,0,0
P00058=0.000,0.000,3.000,0.0000,0.0000,0.0000
///RCONF 1,0,0,0,0,0,0,0,0,0,0,0,0,0,0,0,0,0,0,0,0,0,0,0
P00300=-0.036,-1.505,2.318,0.0000,0.0000,0.0000
P00301=0.046,-2.112,7.779,0.0000,0.0000,0.0000
P00302=-0.180,-2.409,6.326,0.0000,0.0000,0.0000
///RCONF 0,0,0,0,0,0,0,0,0,0,0,0,0,0,0,0,0,0,0,0,0,0,0,0
P00303=-0.004,-1.437,-4.584,0.0000,0.0000,0.0000
P00304=0.028,-1.666,-4.234,0.0000,0.0000,0.0000
P00305=-0.003,-1.920,-3.501,0.0000,0.0000,0.0000
P00306=0.015,-2.252,-3.054,0.0000,0.0000,0.0000
P00307=0.019,-2.151,-5.077,0.0000,0.0000,0.0000
P00308=-0.003,-2.092,-4.888,0.0000,0.0000,0.0000
P00309=-0.040,-2.205,-4.992,0.0000,0.0000,0.0000
P00310=-0.006,-2.490,-5.925,0.0000,0.0000,0.0000
P00311=-0.007,-2.079,-5.307,0.0000,0.0000,0.0000
P00312=-0.032,2.202,-7.632,0.0000,0.0000,0.0000
///RCONF 1,0,0,0,0,0,0,0,0,0,0,0,0,0,0,0,0,0,0,0,0,0,0,0
P00313=-0.088,1.055,2.110,0.0000,0.0000,0.0000
P00314=-0.055,1.752,1.634,0.0000,0.0000,0.0000
P00315=-0.074,0.897,1.645,0.0000,0.0000,0.0000
P00316=0.009,2.112,2.075,0.0000,0.0000,0.0000
P00317=-0.015,2.781,3.126,0.0000,0.0000,0.0000
P00318=-0.086,2.132,2.037,0.0000,0.0000,0.0000
P00319=-0.045,2.990,2.150,0.0000,0.0000,0.0000
///RCONF 0,0,0,0,0,0,0,0,0,0,0,0,0,0,0,0,0,0,0,0,0,0,0,0
P00350=11.519,-0.008,1.149,0.0000,0.0000,0.0000
P00351=13.563,-0.027,-0.653,0.0000,0.0000,0.0000
P00352=13.252,-0.027,-0.827,0.0000,0.0000,0.0000
P00353=10.971,-0.082,0.776,0.0000,0.0000,0.0000
P00354=-0.024,2.508,-1.824,0.0000,0.0000,0.0000
P00355=-0.001,2.528,-1.131,0.0000,0.0000,0.0000
P00356=-0.034,2.921,-0.262,0.0000,0.0000,0.0000
P00357=0.003,3.386,-0.091,0.0000,0.0000,0.0000
P00358=0.014,3.037,-0.020,0.0000,0.0000,0.0000
P00359=-0.005,2.731,0.912,0.0000,0.0000,0.0000
P00360=-0.011,3.412,0.438,0.0000,0.0000,0.0000
P00361=0.018,3.050,1.253,0.0000,0.0000,0.0000
P00401=3.430,-0.021,1.131,0.0000,0.0000,0.0000
P00402=-0.253,1.107,3.062,0.0000,0.0000,0.0000
P00403=-3.666,-0.015,5.328,0.0000,0.0000,0.0000
///RCONF 1,0,0,0,0,0,0,0,0,0,0,0,0,0,0,0,0,0,0,0,0,0,0,0
P00404=0.029,4.189,-1.030,0.0000,0.0000,0.0000
///RCONF 0,0,0,0,0,0,0,0,0,0,0,0,0,0,0,0,0,0,0,0,0,0,0,0
P00405=2.420,0.007,1.427,0.0000,0.0000,0.0000
P00406=3.513,-0.022,0.429,0.0000,0.0000,0.0000
///RCONF 1,0,0,0,1,0,0,0,0,0,0,0,0,0,0,0,0,0,0,0,0,0,0,0
P00407=-0.029,2.348,-1.469,0.0000,0.0000,0.0000
P00408=0.010,1.346,-1.479,0.0000,0.0000,0.0000
///RCONF 1,0,0,0,0,0,0,0,0,0,0,0,0,0,0,0,0,0,0,0,0,0,0,0
P00409=-0.026,2.090,-1.483,0.0000,0.0000,0.0000
P00410=0.001,4.491,-0.583,0.0000,0.0000,0.0000
///RCONF 1,0,0,0,1,0,0,0,0,0,0,0,0,0,0,0,0,0,0,0,0,0,0,0
P00411=-0.015,3.627,0.872,0.0000,0.0000,0.0000
P00412=0.002,3.829,0.787,0.0000,0.0000,0.0000
P00413=0.046,0.107,-0.040,0.0000,0.0000,0.0000
///RCONF 1,0,0,0,0,0,0,0,0,0,0,0,0,0,0,0,0,0,0,0,0,0,0,0
P00414=0.046,0.800,0.739,0.0000,0.0000,0.0000
///RCONF 0,0,0,0,0,0,0,0,0,0,0,0,0,0,0,0,0,0,0,0,0,0,0,0
P00415=-1.781,-1.303,3.250,0.0000,0.0000,0.0000
P00416=0.027,1.119,3.078,0.0000,0.0000,0.0000
///RCONF 1,0,0,0,1,0,0,0,0,0,0,0,0,0,0,0,0,0,0,0,0,0,0,0
P00417=0.059,4.721,3.973,0.0000,0.0000,0.0000
//INST
///DATE 2025/02/21 10:07
///ATTR SC,RW
///GROUP1 RB1,BS1
NOP
CALL JOB:MOVE_INTO_TUNNEL
MOVJ C00000 BC00000 VJ=50.00
MOVJ C00001 BC00001 VJ=40.00
MOVJ C00002 BC00002 VJ=40.00
MOVL C00003 BC00003 V=666.7
MOVJ C00004 BC00004 VJ=30.00
MOVL C00005 BC00005 V=500.0
'------------------------
'W31.2
'------------------------
MOVL C00006 BC00006 V=166.7 PL=0
REFP 3 C00007 BC00007
CALL JOB:SEARCH-R1
SET P0300 P0006
SFTON P0300
MOVL C00008 BC00008 V=166.7 PL=0
REFP 3 C00009 BC00009
CALL JOB:SEARCH-R1
SET P0300 P0006
SFTON P0300
MOVL C00010 BC00010 V=166.7 PL=0
SFTOF
'------------------------
'W31.4
'------------------------
MOVL C00011 BC00011 V=500.0
MOVL C00012 BC00012 V=166.7 PL=0
REFP 3 C00013 BC00013
CALL JOB:SEARCH-R1
SET P0301 P0006
SFTON P0301
MOVL C00014 BC00014 V=166.7 PL=0
REFP 3 C00015 BC00015
CALL JOB:SEARCH-R1
SET P0301 P0006
SFTON P0301
MOVL C00016 BC00016 V=166.7 PL=0
SFTOF
'------------------------
'W31.6
'------------------------
MOVL C00017 BC00017 V=500.0
MOVL C00018 BC00018 V=166.7 PL=0
REFP 3 C00019 BC00019
CALL JOB:SEARCH-R1
SET P0302 P0006
SFTON P0302
MOVL C00020 BC00020 V=166.7 PL=0
REFP 3 C00021 BC00021
CALL JOB:SEARCH-R1
SET P0302 P0006
SFTON P0302
MOVL C00022 BC00022 V=166.7 PL=0
SFTOF
'------------------------
'W31.8
'------------------------
MOVL C00023 BC00023 V=500.0
MOVL C00024 BC00024 V=166.7 PL=0
REFP 3 C00025 BC00025
CALL JOB:SEARCH-R1
SET P0303 P0006
SFTON P0303
MOVL C00026 BC00026 V=166.7 PL=0
REFP 3 C00027 BC00027
CALL JOB:SEARCH-R1
SET P0303 P0006
SFTON P0303
MOVL C00028 BC00028 V=166.7 PL=0
SFTOF
'------------------------
'W31.9
'------------------------
MOVL C00029 BC00029 V=500.0
MOVL C00030 BC00030 V=166.7 PL=0
REFP 3 C00031 BC00031
CALL JOB:SEARCH-R1
SET P0304 P0006
SFTON P0304
MOVL C00032 BC00032 V=166.7 PL=0
REFP 3 C00033 BC00033
CALL JOB:SEARCH-R1
SET P0304 P0006
SFTON P0304
MOVL C00034 BC00034 V=166.7 PL=0
SFTOF
'------------------------
'W31.11
'------------------------
MOVL C00035 BC00035 V=500.0
MOVL C00036 BC00036 V=166.7 PL=0
REFP 3 C00037 BC00037
CALL JOB:SEARCH-R1
SET P0305 P0006
SFTON P0305
MOVL C00038 BC00038 V=166.7 PL=0
REFP 3 C00039 BC00039
CALL JOB:SEARCH-R1
SET P0305 P0006
SFTON P0305
MOVL C00040 BC00040 V=166.7 PL=0
SFTOF
'------------------------
'W31.13
'------------------------
MOVL C00041 BC00041 V=500.0
MOVL C00042 BC00042 V=166.7 PL=0
REFP 3 C00043 BC00043
CALL JOB:SEARCH-R1
SET P0306 P0006
SFTON P0306
MOVL C00044 BC00044 V=166.7 PL=0
REFP 3 C00045 BC00045
CALL JOB:SEARCH-R1
SET P0306 P0006
SFTON P0306
MOVL C00046 BC00046 V=166.7 PL=0
SFTOF
'------------------------
'W31.14
'------------------------
MOVL C00047 BC00047 V=500.0
MOVL C00048 BC00048 V=166.7 PL=0
REFP 3 C00049 BC00049
CALL JOB:SEARCH-R1
SET P0307 P0006
SFTON P0307
MOVL C00050 BC00050 V=166.7 PL=0
REFP 3 C00051 BC00051
CALL JOB:SEARCH-R1
SET P0307 P0006
SFTON P0307
MOVL C00052 BC00052 V=166.7 PL=0
SFTOF
'------------------------
'W31.16
'------------------------
MOVL C00053 BC00053 V=500.0
MOVL C00054 BC00054 V=166.7 PL=0
REFP 3 C00055 BC00055
CALL JOB:SEARCH-R1
SET P0308 P0006
SFTON P0308
MOVL C00056 BC00056 V=166.7 PL=0
REFP 3 C00057 BC00057
CALL JOB:SEARCH-R1
SET P0308 P0006
SFTON P0308
MOVL C00058 BC00058 V=166.7 PL=0
SFTOF
MOVL C00059 BC00059 V=150.0
MOVL C00060 BC00060 V=333.3
MOVL C00061 BC00061 V=500.0
MOVL C00062 BC00062 V=500.0
MOVJ C00063 BC00063 VJ=50.00
MOVL C00064 BC00064 V=666.7
MOVL C00065 BC00065 V=500.0
MOVL C00066 BC00066 V=333.3
'------------------------
'W31.18
'------------------------
MOVL C00067 BC00067 V=133.3 PL=0
REFP 3 C00068 BC00068
CALL JOB:SEARCH-R1
SET P0309 P0006
SFTON P0309
MOVL C00069 BC00069 V=66.7 PL=0
REFP 3 C00070 BC00070
CALL JOB:SEARCH-R1
SET P0309 P0006
SFTON P0309
MOVL C00071 BC00071 V=66.7 PL=0
SFTOF
'------------------------
'W31.19
'------------------------
MOVL C00072 BC00072 V=250.0
MOVL C00073 BC00073 V=166.7 PL=0
REFP 3 C00074 BC00074
CALL JOB:SEARCH-R1
SET P0310 P0006
SFTON P0310
MOVL C00075 BC00075 V=166.7 PL=0
REFP 3 C00076 BC00076
CALL JOB:SEARCH-R1
SET P0310 P0006
SFTON P0310
MOVL C00077 BC00077 V=166.7 PL=0
SFTOF
'------------------------
'W31.21
'------------------------
MOVL C00078 BC00078 V=500.0
MOVL C00079 BC00079 V=166.7 PL=0
REFP 3 C00080 BC00080
CALL JOB:SEARCH-R1
SET P0311 P0006
SFTON P0311
MOVL C00081 BC00081 V=166.7 PL=0
REFP 3 C00082 BC00082
CALL JOB:SEARCH-R1
SET P0311 P0006
SFTON P0311
MOVL C00083 BC00083 V=166.7 PL=0
SFTOF
'------------------------
'W31.22
'------------------------
MOVL C00084 BC00084 V=500.0
MOVL C00085 BC00085 V=166.7 PL=0
REFP 3 C00086 BC00086
CALL JOB:SEARCH-R1
SET P0312 P0006
SFTON P0312
MOVL C00087 BC00087 V=166.7 PL=0
REFP 3 C00088 BC00088
CALL JOB:SEARCH-R1
SET P0312 P0006
SFTON P0312
MOVL C00089 BC00089 V=166.7 PL=0
SFTOF
'------------------------
'W31.24
'------------------------
MOVL C00090 BC00090 V=500.0
MOVL C00091 BC00091 V=166.7 PL=0
REFP 3 C00092 BC00092
CALL JOB:SEARCH-R1
SET P0313 P0006
SFTON P0313
MOVL C00093 BC00093 V=166.7 PL=0
REFP 3 C00094 BC00094
CALL JOB:SEARCH-R1
SET P0313 P0006
SFTON P0313
MOVL C00095 BC00095 V=166.7 PL=0
SFTOF
'------------------------
'W31.26
'------------------------
MOVL C00096 BC00096 V=500.0
MOVL C00097 BC00097 V=166.7 PL=0
REFP 3 C00098 BC00098
CALL JOB:SEARCH-R1
SET P0314 P0006
SFTON P0314
MOVL C00099 BC00099 V=166.7 PL=0
REFP 3 C00100 BC00100
CALL JOB:SEARCH-R1
SET P0314 P0006
SFTON P0314
MOVL C00101 BC00101 V=166.7 PL=0
SFTOF
'------------------------
'W31.27
'------------------------
MOVL C00102 BC00102 V=500.0
MOVL C00103 BC00103 V=166.7 PL=0
REFP 3 C00104 BC00104
CALL JOB:SEARCH-R1
SET P0315 P0006
SFTON P0315
MOVL C00105 BC00105 V=166.7 PL=0
REFP 3 C00106 BC00106
CALL JOB:SEARCH-R1
SET P0315 P0006
SFTON P0315
MOVL C00107 BC00107 V=166.7 PL=0
SFTOF
MOVL C00108 BC00108 V=333.3
MOVL C00109 BC00109 V=166.7 PL=0
REFP 3 C00110 BC00110
CALL JOB:SEARCH-R1
SET P0316 P0006
SFTON P0316
MOVL C00111 BC00111 V=166.7 PL=0
REFP 3 C00112 BC00112
CALL JOB:SEARCH-R1
SET P0316 P0006
SFTON P0316
MOVL C00113 BC00113 V=166.7 PL=0
SFTOF
MOVL C00114 BC00114 V=333.3
MOVL C00115 BC00115 V=666.7
MOVL C00116 BC00116 V=666.7
MOVL C00117 BC00117 V=666.7
MOVL C00118 BC00118 V=666.7
MOVL C00119 BC00119 V=666.7
MOVL C00120 BC00120 V=666.7
MOVL C00121 BC00121 V=250.0
'------------------------
'W31.29
'------------------------
'------------------------
'W31.31
'------------------------
MOVL C00122 BC00122 V=500.0
MOVL C00123 BC00123 V=166.7 PL=0
REFP 3 C00124 BC00124
CALL JOB:SEARCH-R1
SET P0317 P0006
SFTON P0317
MOVL C00125 BC00125 V=166.7 PL=0
REFP 3 C00126 BC00126
CALL JOB:SEARCH-R1
SET P0317 P0006
SFTON P0317
MOVL C00127 BC00127 V=166.7 PL=0
SFTOF
'------------------------
'W31.32
'------------------------
MOVL C00128 BC00128 V=250.0
MOVL C00129 BC00129 V=166.7 PL=0
REFP 3 C00130 BC00130
CALL JOB:SEARCH-R1
SET P0318 P0006
SFTON P0318
MOVL C00131 BC00131 V=166.7 PL=0
REFP 3 C00132 BC00132
CALL JOB:SEARCH-R1
SET P0318 P0006
SFTON P0318
MOVL C00133 BC00133 V=166.7 PL=0
SFTOF
MOVL C00134 BC00134 V=333.3
MOVL C00135 BC00135 V=333.3
MOVL C00136 BC00136 V=166.7 PL=0
REFP 3 C00137 BC00137
CALL JOB:SEARCH-R1
SET P0319 P0006
SFTON P0319
MOVL C00138 BC00138 V=166.7 PL=0
REFP 3 C00139 BC00139
CALL JOB:SEARCH-R1
SET P0319 P0006
SFTON P0319
MOVL C00140 BC00140 V=166.7 PL=0
SFTOF
MOVL C00141 BC00141 V=250.0
MOVL C00142 BC00142 V=333.3
MOVL C00143 BC00143 V=333.3
MOVL C00144 BC00144 V=666.7
MOVJ C00145 BC00145 VJ=50.00
MOVJ C00146 BC00146 VJ=50.00
MOVJ C00147 BC00147 VJ=30.00
MOVL C00148 BC00148 V=166.7
'------------------------
'W214B L
'------------------------
MOVL C00149 BC00149 V=166.7 PL=0
REFP 3 C00150 BC00150
CALL JOB:SEARCH-R1
IMOV P0058 V=16.7
SET P0350 P0006
SFTON P0350
REFP 3 C00151 BC00151
CALL JOB:SEARCH-R1
SET P0350 P0006
SFTON P0350
MOVL C00152 BC00152 V=166.7 PL=0
SFTOF
'------------------------
'W214A P
'------------------------
MOVJ C00153 BC00153 VJ=40.00
MOVL C00154 BC00154 V=166.7 PL=0
REFP 3 C00155 BC00155
CALL JOB:SEARCH-R1
IMOV P0058 V=16.7
SET P0351 P0006
SFTON P0351
REFP 3 C00156 BC00156
CALL JOB:SEARCH-R1
SET P0351 P0006
SFTON P0351
MOVL C00157 BC00157 V=166.7 PL=0
SFTOF
'------------------------
'W219B L
'------------------------
MOVJ C00158 BC00158 VJ=40.00
MOVL C00159 BC00159 V=166.7 PL=0
REFP 3 C00160 BC00160
CALL JOB:SEARCH-R1
IMOV P0058 V=16.7
SET P0352 P0006
SFTON P0352
REFP 3 C00161 BC00161
CALL JOB:SEARCH-R1
SET P0352 P0006
SFTON P0352
MOVL C00162 BC00162 V=166.7 PL=0
SFTOF
'------------------------
'W219B P
'------------------------
MOVJ C00163 BC00163 VJ=40.00
MOVL C00164 BC00164 V=166.7 PL=0
REFP 3 C00165 BC00165
CALL JOB:SEARCH-R1
IMOV P0058 V=16.7
SET P0353 P0006
SFTON P0353
REFP 3 C00166 BC00166
CALL JOB:SEARCH-R1
SET P0353 P0006
SFTON P0353
MOVL C00167 BC00167 V=166.7 PL=0
SFTOF
'------------------------
'W213B L
'------------------------
MOVJ C00168 BC00168 VJ=40.00
MOVL C00169 BC00169 V=166.7 PL=0
REFP 3 C00170 BC00170
CALL JOB:SEARCH-R1
IMOV P0058 V=16.7
SET P0354 P0006
SFTON P0354
REFP 3 C00171 BC00171
CALL JOB:SEARCH-R1
SET P0354 P0006
SFTON P0354
MOVL C00172 BC00172 V=166.7 PL=0
SFTOF
'------------------------
'W213B P
'------------------------
MOVJ C00173 BC00173 VJ=40.00
MOVL C00174 BC00174 V=166.7 PL=0
REFP 3 C00175 BC00175
CALL JOB:SEARCH-R1
IMOV P0058 V=16.7
SET P0355 P0006
SFTON P0355
REFP 3 C00176 BC00176
CALL JOB:SEARCH-R1
SET P0355 P0006
SFTON P0355
MOVL C00177 BC00177 V=166.7 PL=0
SFTOF
'------------------------
'W218B L
'------------------------
MOVJ C00178 BC00178 VJ=40.00
MOVL C00179 BC00179 V=166.7 PL=0
REFP 3 C00180 BC00180
CALL JOB:SEARCH-R1
IMOV P0058 V=16.7
SET P0356 P0006
SFTON P0356
REFP 3 C00181 BC00181
CALL JOB:SEARCH-R1
SET P0356 P0006
SFTON P0356
MOVL C00182 BC00182 V=166.7 PL=0
SFTOF
'------------------------
'W218B P
'------------------------
MOVJ C00183 BC00183 VJ=40.00
MOVL C00184 BC00184 V=166.7 PL=0
REFP 3 C00185 BC00185
CALL JOB:SEARCH-R1
IMOV P0058 V=16.7
SET P0357 P0006
SFTON P0357
REFP 3 C00186 BC00186
CALL JOB:SEARCH-R1
SET P0357 P0006
SFTON P0357
MOVL C00187 BC00187 V=166.7 PL=0
SFTOF
'------------------------
'W215B L
'------------------------
MOVJ C00188 BC00188 VJ=40.00
MOVL C00189 BC00189 V=166.7 PL=0
REFP 3 C00190 BC00190
CALL JOB:SEARCH-R1
IMOV P0058 V=16.7
SET P0358 P0006
SFTON P0358
REFP 3 C00191 BC00191
CALL JOB:SEARCH-R1
SET P0358 P0006
SFTON P0358
MOVL C00192 BC00192 V=166.7 PL=0
SFTOF
'------------------------
'W215B P
'------------------------
MOVL C00193 BC00193 V=666.7
MOVL C00194 BC00194 V=166.7 PL=0
REFP 3 C00195 BC00195
CALL JOB:SEARCH-R1
IMOV P0058 V=16.7
SET P0359 P0006
SFTON P0359
REFP 3 C00196 BC00196
CALL JOB:SEARCH-R1
SET P0359 P0006
SFTON P0359
MOVL C00197 BC00197 V=166.7 PL=0
SFTOF
'------------------------
'W217B L
'------------------------
MOVL C00198 BC00198 V=666.7
MOVL C00199 BC00199 V=166.7 PL=0
REFP 3 C00200 BC00200
CALL JOB:SEARCH-R1
IMOV P0058 V=16.7
SET P0360 P0006
SFTON P0360
REFP 3 C00201 BC00201
CALL JOB:SEARCH-R1
SET P0360 P0006
SFTON P0360
MOVL C00202 BC00202 V=166.7 PL=0
SFTOF
'------------------------
'W217B P
'------------------------
MOVL C00203 BC00203 V=666.7
MOVL C00204 BC00204 V=166.7 PL=0
REFP 3 C00205 BC00205
CALL JOB:SEARCH-R1
IMOV P0058 V=16.7
SET P0361 P0006
SFTON P0361
REFP 3 C00206 BC00206
CALL JOB:SEARCH-R1
SET P0361 P0006
SFTON P0361
MOVL C00207 BC00207 V=166.7 PL=0
SFTOF
MOVL C00208 BC00208 V=333.3
MOVL C00209 BC00209 V=666.7
MOVL C00210 BC00210 V=666.7
MOVJ C00211 BC00211 VJ=50.00
MOVJ C00212 BC00212 VJ=50.00
COMM MOVJ C00213 BC00213 VJ=40.00
COMM MOVJ C00214 BC00214 VJ=40.00
COMM MOVJ C00215 BC00215 VJ=25.00
COMM MOVJ C00216 BC00216 VJ=30.00
COMM MOVJ C00217 BC00217 VJ=30.00
COMM MOVJ C00218 BC00218 VJ=20.00
COMM MOVL C00219 BC00219 V=500.0
COMM '------------------------
COMM 'W27.4
COMM '------------------------
COMM MOVL C00220 BC00220 V=166.7 PL=0
COMM REFP 3 C00221 BC00221
COMM CALL JOB:SEARCH-R1
COMM SET P0401 P0006
COMM SFTON P0401
COMM MOVL C00222 BC00222 V=166.7 PL=0
COMM REFP 3 C00223 BC00223
COMM CALL JOB:SEARCH-R1
COMM SET P0401 P0006
COMM SFTON P0401
COMM MOVL C00224 BC00224 V=166.7 PL=0
COMM SFTOF
COMM '------------------------
COMM 'W27.6
COMM '------------------------
COMM MOVL C00225 BC00225 V=666.7
COMM MOVL C00226 BC00226 V=166.7 PL=0
COMM REFP 3 C00227 BC00227
COMM CALL JOB:SEARCH-R1
COMM SET P0402 P0006
COMM SFTON P0402
COMM MOVL C00228 BC00228 V=166.7 PL=0
COMM REFP 3 C00229 BC00229
COMM CALL JOB:SEARCH-R1
COMM SET P0402 P0006
COMM SFTON P0402
COMM MOVL C00230 BC00230 V=166.7 PL=0
COMM SFTOF
COMM MOVL C00231 BC00231 V=500.0
COMM MOVL C00232 BC00232 V=500.0
COMM '------------------------
COMM 'W27.8
COMM '------------------------
COMM MOVL C00233 BC00233 V=333.3
COMM MOVL C00234 BC00234 V=166.7 PL=0
COMM REFP 3 C00235 BC00235
COMM CALL JOB:SEARCH-R1
COMM SET P0403 P0006
COMM SFTON P0403
COMM MOVL C00236 BC00236 V=166.7 PL=0
COMM REFP 3 C00237 BC00237
COMM CALL JOB:SEARCH-R1
COMM SET P0403 P0006
COMM SFTON P0403
COMM MOVL C00238 BC00238 V=166.7 PL=0
COMM SFTOF
COMM MOVJ C00239 BC00239 VJ=25.00
COMM MOVJ C00240 BC00240 VJ=25.00
COMM MOVJ C00241 BC00241 VJ=30.00
COMM MOVJ C00242 BC00242 VJ=40.00
COMM MOVJ C00243 BC00243 VJ=30.00
COMM '------------------------
COMM 'W27.9
COMM '------------------------
COMM MOVL C00244 BC00244 V=500.0
COMM MOVL C00245 BC00245 V=166.7 PL=0
COMM REFP 3 C00246 BC00246
COMM CALL JOB:SEARCH-R1
COMM SET P0404 P0006
COMM SFTON P0404
COMM MOVL C00247 BC00247 V=166.7 PL=0
COMM REFP 3 C00248 BC00248
COMM CALL JOB:SEARCH-R1
COMM SET P0404 P0006
COMM SFTON P0404
COMM MOVL C00249 BC00249 V=166.7 PL=0
COMM SFTOF
COMM MOVL C00250 BC00250 V=500.0
COMM '------------------------
COMM 'W27.11
COMM '------------------------
COMM MOVL C00251 BC00251 V=500.0
COMM MOVL C00252 BC00252 V=166.7 PL=0
COMM REFP 3 C00253 BC00253
COMM CALL JOB:SEARCH-R1
COMM SET P0405 P0006
COMM SFTON P0405
COMM MOVL C00254 BC00254 V=166.7 PL=0
COMM REFP 3 C00255 BC00255
COMM CALL JOB:SEARCH-R1
COMM SET P0405 P0006
COMM SFTON P0405
COMM MOVL C00256 BC00256 V=166.7 PL=0
COMM SFTOF
COMM MOVL C00257 BC00257 V=666.7
COMM MOVL C00258 BC00258 V=666.7
COMM '------------------------
COMM 'W27.13
COMM '------------------------
COMM MOVL C00259 BC00259 V=333.3
COMM MOVL C00260 BC00260 V=166.7 PL=0
COMM REFP 3 C00261 BC00261
COMM CALL JOB:SEARCH-R1
COMM SET P0406 P0006
COMM SFTON P0406
COMM MOVL C00262 BC00262 V=166.7 PL=0
COMM REFP 3 C00263 BC00263
COMM CALL JOB:SEARCH-R1
COMM SET P0406 P0006
COMM SFTON P0406
COMM MOVL C00264 BC00264 V=166.7 PL=0
COMM SFTOF
COMM '------------------------
COMM 'W27.14
COMM '------------------------
COMM MOVL C00265 BC00265 V=666.7
COMM MOVL C00266 BC00266 V=166.7 PL=0
COMM REFP 3 C00267 BC00267
COMM CALL JOB:SEARCH-R1
COMM SET P0407 P0006
COMM SFTON P0407
COMM MOVL C00268 BC00268 V=166.7 PL=0
COMM REFP 3 C00269 BC00269
COMM CALL JOB:SEARCH-R1
COMM SET P0407 P0006
COMM SFTON P0407
COMM MOVL C00270 BC00270 V=166.7 PL=0
COMM SFTOF
COMM MOVL C00271 BC00271 V=666.7
COMM '------------------------
COMM 'W27.16
COMM '------------------------
COMM MOVL C00272 BC00272 V=333.3
COMM MOVL C00273 BC00273 V=166.7 PL=0
COMM REFP 3 C00274 BC00274
COMM CALL JOB:SEARCH-R1
COMM SET P0408 P0006
COMM SFTON P0408
COMM MOVL C00275 BC00275 V=166.7 PL=0
COMM REFP 3 C00276 BC00276
COMM CALL JOB:SEARCH-R1
COMM SET P0408 P0006
COMM SFTON P0408
COMM MOVL C00277 BC00277 V=166.7 PL=0
COMM SFTOF
COMM MOVL C00278 BC00278 V=666.7
COMM MOVJ C00279 BC00279 VJ=30.00
COMM MOVJ C00280 BC00280 VJ=50.00
COMM MOVJ C00281 BC00281 VJ=40.00
COMM MOVJ C00282 BC00282 VJ=30.00
COMM '------------------------
COMM 'W27.18
COMM '------------------------
COMM MOVL C00283 BC00283 V=333.3
COMM MOVL C00284 BC00284 V=166.7 PL=0
COMM REFP 3 C00285 BC00285
COMM CALL JOB:SEARCH-R1
COMM SET P0409 P0006
COMM SFTON P0409
COMM MOVL C00286 BC00286 V=166.7 PL=0
COMM REFP 3 C00287 BC00287
COMM CALL JOB:SEARCH-R1
COMM SET P0409 P0006
COMM SFTON P0409
COMM MOVL C00288 BC00288 V=166.7 PL=0
COMM SFTOF
COMM '------------------------
COMM 'W27.19
COMM '------------------------
COMM MOVL C00289 BC00289 V=666.7
COMM MOVL C00290 BC00290 V=166.7 PL=0
COMM REFP 3 C00291 BC00291
COMM CALL JOB:SEARCH-R1
COMM SET P0410 P0006
COMM SFTON P0410
COMM MOVL C00292 BC00292 V=166.7 PL=0
COMM REFP 3 C00293 BC00293
COMM CALL JOB:SEARCH-R1
COMM SET P0410 P0006
COMM SFTON P0410
COMM MOVL C00294 BC00294 V=166.7 PL=0
COMM SFTOF
COMM MOVL C00295 BC00295 V=666.7
COMM '------------------------
COMM 'W27.21
COMM '------------------------
COMM MOVL C00296 BC00296 V=166.7 PL=0
COMM REFP 3 C00297 BC00297
COMM CALL JOB:SEARCH-R1
COMM SET P0411 P0006
COMM SFTON P0411
COMM MOVL C00298 BC00298 V=166.7 PL=0
COMM REFP 3 C00299 BC00299
COMM CALL JOB:SEARCH-R1
COMM SET P0411 P0006
COMM SFTON P0411
COMM MOVL C00300 BC00300 V=166.7 PL=0
COMM SFTOF
COMM '------------------------
COMM 'W27.22
COMM '------------------------
COMM MOVL C00301 BC00301 V=666.7
COMM MOVL C00302 BC00302 V=166.7 PL=0
COMM REFP 3 C00303 BC00303
COMM CALL JOB:SEARCH-R1
COMM SET P0412 P0006
COMM SFTON P0412
COMM MOVL C00304 BC00304 V=166.7 PL=0
COMM REFP 3 C00305 BC00305
COMM CALL JOB:SEARCH-R1
COMM SET P0412 P0006
COMM SFTON P0412
COMM MOVL C00306 BC00306 V=166.7 PL=0
COMM SFTOF
COMM MOVL C00307 BC00307 V=666.7
COMM MOVJ C00308 BC00308 VJ=30.00
COMM MOVL C00309 BC00309 V=500.0
COMM '------------------------
COMM 'W27.24
COMM '------------------------
COMM MOVL C00310 BC00310 V=666.7
COMM MOVL C00311 BC00311 V=166.7 PL=0
COMM REFP 3 C00312 BC00312
COMM CALL JOB:SEARCH-R1
COMM SET P0413 P0006
COMM SFTON P0413
COMM MOVL C00313 BC00313 V=166.7 PL=0
COMM REFP 3 C00314 BC00314
COMM CALL JOB:SEARCH-R1
COMM SET P0413 P0006
COMM SFTON P0413
COMM MOVL C00315 BC00315 V=166.7 PL=0
COMM SFTOF
COMM MOVL C00316 BC00316 V=666.7
COMM MOVJ C00317 BC00317 VJ=50.00
COMM MOVJ C00318 BC00318 VJ=50.00
COMM MOVJ C00319 BC00319 VJ=50.00
COMM MOVJ C00320 BC00320 VJ=20.00
COMM MOVJ C00321 BC00321 VJ=10.00
COMM '------------------------
COMM 'W27.26
COMM '------------------------
COMM MOVL C00322 BC00322 V=333.3
COMM MOVL C00323 BC00323 V=166.7 PL=0
COMM REFP 3 C00324 BC00324
COMM CALL JOB:SEARCH-R1
COMM SET P0414 P0006
COMM SFTON P0414
COMM MOVL C00325 BC00325 V=166.7 PL=0
COMM REFP 3 C00326 BC00326
COMM CALL JOB:SEARCH-R1
COMM SET P0414 P0006
COMM SFTON P0414
COMM MOVL C00327 BC00327 V=166.7 PL=0
COMM SFTOF
COMM MOVL C00328 BC00328 V=333.3
COMM MOVJ C00329 BC00329 VJ=30.00
COMM MOVJ C00330 BC00330 VJ=30.00
COMM MOVJ C00331 BC00331 VJ=30.00
COMM GETE D040 P0414 (1)
COMM GETE D041 P0414 (2)
COMM GETE D042 P0414 (3)
COMM SETE P0415 (1) D040
COMM SETE P0415 (2) D041
COMM SETE P0415 (3) D042
COMM '------------------------
COMM 'W27.29
COMM '------------------------
COMM MOVJ C00332 BC00332 VJ=30.00
COMM MOVJ C00333 BC00333 VJ=30.00
COMM MOVL C00334 BC00334 V=333.3
COMM MOVL C00335 BC00335 V=166.7 PL=0
COMM REFP 3 C00336 BC00336
COMM CALL JOB:SEARCH-R1
COMM SET P0416 P0006
COMM SFTON P0416
COMM MOVL C00337 BC00337 V=166.7 PL=0
COMM REFP 3 C00338 BC00338
COMM CALL JOB:SEARCH-R1
COMM SET P0416 P0006
COMM SFTON P0416
COMM MOVL C00339 BC00339 V=166.7 PL=0
COMM SFTOF
COMM '------------------------
COMM 'W27.31
COMM '------------------------
COMM MOVL C00340 BC00340 V=666.7
COMM MOVL C00341 BC00341 V=166.7 PL=0
COMM REFP 3 C00342 BC00342
COMM CALL JOB:SEARCH-R1
COMM SET P0417 P0006
COMM SFTON P0417
COMM MOVL C00343 BC00343 V=166.7 PL=0
COMM REFP 3 C00344 BC00344
COMM CALL JOB:SEARCH-R1
COMM SET P0417 P0006
COMM SFTON P0417
COMM MOVL C00345 BC00345 V=166.7 PL=0
COMM SFTOF
COMM '------------------------
COMM 'W27.32
COMM '------------------------
COMM MOVL C00346 BC00346 V=333.3
MOVJ C00347 BC00347 VJ=50.00
CALL JOB:FRONT_SEARCH_-90ST-1_5540
MOVJ C00348 BC00348 VJ=50.00
MOVJ C00349 BC00349 VJ=50.00
MOVJ C00350 BC00350 VJ=50.00
MOVL C00351 BC00351 V=666.7
MOVJ C00352 BC00352 VJ=30.00
'------------------------
'W31.2
'------------------------
SFTON P0300
MOVL C00353 BC00353 V=333.3
MOVL C00354 BC00354 V=166.7 PL=0
MACRO1 MJ#(0) ARGF10
ARCON
MOVL C00355 BC00355 V=10.8
ARCOF
MOVL C00356 BC00356 V=166.7
SFTOF
'------------------------
'W31.4
'------------------------
SFTON P0301
MOVL C00357 BC00357 V=666.7
MOVL C00358 BC00358 V=166.7 PL=0
ARCON
MOVL C00359 BC00359 V=10.8
ARCOF
MOVL C00360 BC00360 V=166.7
SFTOF
'------------------------
'W31.6
'------------------------
SFTON P0302
MOVL C00361 BC00361 V=666.7
MOVL C00362 BC00362 V=166.7 PL=0
ARCON
MOVL C00363 BC00363 V=10.8
ARCOF
MOVL C00364 BC00364 V=166.7
SFTOF
'------------------------
'W31.8
'------------------------
SFTON P0303
MOVL C00365 BC00365 V=666.7
MOVL C00366 BC00366 V=166.7 PL=0
ARCON
MOVL C00367 BC00367 V=10.8
ARCOF
MOVL C00368 BC00368 V=166.7
SFTOF
'------------------------
'W31.9
'------------------------
SFTON P0304
MOVL C00369 BC00369 V=666.7
MOVL C00370 BC00370 V=166.7 PL=0
ARCON
MOVL C00371 BC00371 V=10.8
ARCOF
MOVL C00372 BC00372 V=166.7
SFTOF
MOVL C00373 BC00373 V=500.0
MOVL C00374 BC00374 V=500.0
MOVJ C00375 BC00375 VJ=50.00
MOVJ C00376 BC00376 VJ=50.00
COMM '::::::::::::::::::::::::::::::::
COMM '::::::::::::::::::::::::::::::::
COMM '::::::::::::::::::::::::::::::::
COMM '::::::::::::::::::::::::::::::::
COMM '::::::::::::::::::::::::::::::::
COMM MOVJ C00377 BC00377 VJ=40.00
COMM MOVJ C00378 BC00378 VJ=40.00
COMM MOVJ C00379 BC00379 VJ=40.00
COMM MOVJ C00380 BC00380 VJ=40.00
COMM MOVJ C00381 BC00381 VJ=40.00
COMM MOVJ C00382 BC00382 VJ=40.00
COMM '------------------------
COMM 'W27.2
COMM '------------------------
COMM MOVL C00383 BC00383 V=500.0
COMM SFTON P0401
COMM MOVL C00384 BC00384 V=166.7 PL=0
COMM MACRO1 MJ#(0) ARGF24
COMM ARCON
COMM MOVL C00385 BC00385 V=7.5
COMM ARCOF
COMM SFTOF
COMM 'BELKA PRZEJAZD
COMM MOVL C00386 BC00386 V=500.0
COMM '------------------------
COMM 'W27.6
COMM '------------------------
COMM SFTON P0402
COMM MOVL C00387 BC00387 V=500.0
COMM MOVL C00388 BC00388 V=166.7 PL=0
COMM MACRO1 MJ#(0) ARGF24
COMM ARCON
COMM MOVL C00389 BC00389 V=7.5
COMM ARCOF
COMM MOVL C00390 BC00390 V=166.7
COMM SFTOF
COMM MOVJ C00391 BC00391 VJ=20.00
COMM '------------------------
COMM 'W27.8
COMM '------------------------
COMM SFTON P0403
COMM MOVL C00392 BC00392 V=500.0
COMM MOVL C00393 BC00393 V=166.7 PL=0
COMM MACRO1 MJ#(0) ARGF24
COMM ARCON
COMM MOVL C00394 BC00394 V=7.5
COMM ARCOF
COMM MOVL C00395 BC00395 V=166.7
COMM SFTOF
COMM MOVL C00396 BC00396 V=500.0
COMM MOVJ C00397 BC00397 VJ=50.00
MOVJ C00398 BC00398 VJ=50.00
MOVJ C00399 BC00399 VJ=50.00
MOVJ C00400 BC00400 VJ=50.00
MOVL C00401 BC00401 V=666.7
'------------------------
'W213A
'------------------------
SFTON P0355
MOVL C00402 BC00402 V=666.7
MOVL C00403 BC00403 V=166.7 PL=0
MACRO1 MJ#(0) ARGF9
ARCON
SFTOF
SFTON P0354
MOVL C00404 BC00404 V=11.2
ARCOF
MOVL C00405 BC00405 V=333.3
SFTOF
MOVJ C00406 BC00406 VJ=50.00
MOVJ C00407 BC00407 VJ=50.00
MOVJ C00408 BC00408 VJ=30.00
MOVJ C00409 BC00409 VJ=20.00
MOVJ C00410 BC00410 VJ=20.00
'5.5.1
'------------------------
'W31.11
'------------------------
SFTON P0305
MOVL C00411 BC00411 V=333.3
MOVL C00412 BC00412 V=166.7 PL=0
MACRO1 MJ#(0) ARGF10
ARCON
MOVL C00413 BC00413 V=10.8
ARCOF
MOVL C00414 BC00414 V=166.7
SFTOF
'------------------------
'W31.13
'------------------------
SFTON P0306
MOVL C00415 BC00415 V=500.0
'SPR CZY W DOBRYM MIEJSCU SPOINA
MOVL C00416 BC00416 V=166.7 PL=0
ARCON
MOVL C00417 BC00417 V=10.8
ARCOF
MOVL C00418 BC00418 V=166.7
SFTOF
'------------------------
'W31.14
'------------------------
SFTON P0307
MOVL C00419 BC00419 V=333.3
MOVL C00420 BC00420 V=166.7 PL=0
ARCON
MOVL C00421 BC00421 V=8.3
ARCOF
MOVL C00422 BC00422 V=166.7
SFTOF
MOVL C00423 BC00423 V=333.3
MOVL C00424 BC00424 V=500.0
MOVJ C00425 BC00425 VJ=30.00
MOVJ C00426 BC00426 VJ=30.00
MOVJ C00427 BC00427 VJ=30.00
MOVJ C00428 BC00428 VJ=50.00
COMM '::::::::::::::::::::::::::::::::
COMM '::::::::::::::::::::::::::::::::
COMM '------------------------
COMM 'W27.9
COMM '------------------------
COMM '::::::::::::::::::::::::::::::::
COMM '::::::::::::::::::::::::::::::::
COMM MOVJ C00429 BC00429 VJ=25.00
COMM MOVJ C00430 BC00430 VJ=40.00
COMM SFTON P0404
COMM MOVL C00431 BC00431 V=500.0
COMM MOVL C00432 BC00432 V=166.7 PL=0
COMM MACRO1 MJ#(0) ARGF24
COMM ARCON
COMM MOVL C00433 BC00433 V=7.5
COMM ARCOF
COMM MOVL C00434 BC00434 V=166.7
COMM SFTOF
COMM '------------------------
COMM 'W27.11
COMM '------------------------
COMM SFTON P0406
COMM MOVL C00435 BC00435 V=666.7
COMM MOVL C00436 BC00436 V=166.7 PL=0
COMM MACRO1 MJ#(0) ARGF24
COMM ARCON
COMM MOVL C00437 BC00437 V=7.5
COMM ARCOF
COMM MOVL C00438 BC00438 V=166.7
COMM SFTOF
COMM '------------------------
COMM 'W27.13
'------------------------
COMM SFTON P0406
COMM MOVL C00439 BC00439 V=666.7
COMM MOVL C00440 BC00440 V=166.7 PL=0
COMM MACRO1 MJ#(0) ARGF24
COMM ARCON
COMM MOVL C00441 BC00441 V=7.5
COMM ARCOF
COMM MOVL C00442 BC00442 V=166.7
COMM SFTOF
COMM MOVJ C00443 BC00443 VJ=40.00
COMM MOVJ C00444 BC00444 VJ=50.00
COMM MOVJ C00445 BC00445 VJ=50.00
COMM MOVJ C00446 BC00446 VJ=50.00
MOVJ C00447 BC00447 VJ=50.00
'::::::::::::::::::::::::
'::::::::::::::::::::::::
'::::::::::::::::::::::::
'::::::::::::::::::::::::
'::::::::::::::::::::::::
'::::::::::::::::::::::::
'::::::::::::::::::::::::
MOVJ C00448 BC00448 VJ=50.00
MOVJ C00449 BC00449 VJ=50.00
'------------------------
'W214A
'------------------------
SFTON P0351
MOVL C00450 BC00450 V=500.0
MOVL C00451 BC00451 V=166.7 PL=0
MACRO1 MJ#(0) ARGF9
ARCON
SFTOF
SFTON P0350
MOVL C00452 BC00452 V=11.7
ARCOF
MOVL C00453 BC00453 V=333.3
SFTOF
MOVJ C00454 BC00454 VJ=50.00
MOVJ C00455 BC00455 VJ=50.00
MOVJ C00456 BC00456 VJ=50.00
MOVJ C00457 BC00457 VJ=40.00
MOVJ C00458 BC00458 VJ=50.00
MOVJ C00459 BC00459 VJ=30.00
MOVJ C00460 BC00460 VJ=30.00
MOVJ C00461 BC00461 VJ=30.00
MOVJ C00462 BC00462 VJ=30.00
'------------------------
'W31.16
'------------------------
SFTON P0308
MOVL C00463 BC00463 V=666.7
MOVL C00464 BC00464 V=166.7 PL=0
MACRO1 MJ#(0) ARGF10
ARCON
MOVL C00465 BC00465 V=10.8
ARCOF
MOVL C00466 BC00466 V=166.7
SFTOF
MOVL C00467 BC00467 V=333.3
SFTON P0309
MOVL C00468 BC00468 V=166.7
ARCON
MOVL C00469 BC00469 V=10.8
ARCOF
SFTOF
MOVL C00470 BC00470 V=250.0
MOVL C00471 BC00471 V=666.7
MOVL C00472 BC00472 V=666.7
MOVL C00473 BC00473 V=666.7
MOVL C00474 BC00474 V=833.3
MOVL C00475 BC00475 V=666.7
'------------------------
'W31.19
'------------------------
SFTON P0310
MOVL C00476 BC00476 V=333.3
MOVL C00477 BC00477 V=166.7 PL=0
ARCON
MOVL C00478 BC00478 V=10.8
ARCOF
MOVL C00479 BC00479 V=166.7
SFTOF
MOVL C00480 BC00480 V=500.0
MOVL C00481 BC00481 V=666.7
MOVL C00482 BC00482 V=666.7
MOVJ C00483 BC00483 VJ=40.00
MOVJ C00484 BC00484 VJ=40.00
COMM '::::::::::::::::::::::::
COMM '::::::::::::::::::::::::
COMM '::::::::::::::::::::::::
COMM '::::::::::::::::::::::::
COMM '::::::::::::::::::::::::
COMM '::::::::::::::::::::::::
COMM '::::::::::::::::::::::::
COMM MOVJ C00485 BC00485 VJ=50.00
COMM MOVJ C00486 BC00486 VJ=30.00
COMM '::::::::::::::::::::::::::::::::
COMM '::::::::::::::::::::::::::::::::
COMM '------------------------
COMM 'W27.14
COMM '------------------------
COMM '::::::::::::::::::::::::::::::::
COMM '::::::::::::::::::::::::::::::::
COMM MOVL C00487 BC00487 V=500.0
COMM MOVL C00488 BC00488 V=500.0
COMM SFTON P0407
COMM MOVL C00489 BC00489 V=166.7 PL=0
COMM MACRO1 MJ#(0) ARGF24
COMM ARCON
COMM MOVL C00490 BC00490 V=7.5
COMM ARCOF
COMM MOVL C00491 BC00491 V=166.7
COMM SFTOF
COMM MOVJ C00492 BC00492 VJ=30.00
COMM '------------------------
COMM 'W27.16
COMM '------------------------
COMM SFTON P0408
COMM MOVL C00493 BC00493 V=500.0
COMM MOVL C00494 BC00494 V=166.7 PL=0
COMM MACRO1 MJ#(0) ARGF24
COMM ARCON
COMM MOVL C00495 BC00495 V=6.7
COMM ARCOF
COMM MOVL C00496 BC00496 V=166.7
COMM MOVL C00497 BC00497 V=666.7
COMM MOVJ C00498 BC00498 VJ=50.00
COMM SFTOF
COMM '------------------------
COMM 'W27.18
COMM '------------------------
COMM SFTON P0409
COMM MOVL C00499 BC00499 V=500.0
COMM MOVL C00500 BC00500 V=166.7 PL=0
COMM MACRO1 MJ#(0) ARGF24
COMM ARCON
COMM MOVL C00501 BC00501 V=7.5
COMM ARCOF
COMM MOVL C00502 BC00502 V=166.7
COMM SFTOF
COMM MOVJ C00503 BC00503 VJ=30.00
COMM MOVJ C00504 BC00504 VJ=30.00
COMM MOVJ C00505 BC00505 VJ=40.00
MOVJ C00506 BC00506 VJ=50.00
'::::::::::::::::::::::::
'::::::::::::::::::::::::
'::::::::::::::::::::::::
'::::::::::::::::::::::::
'::::::::::::::::::::::::
'::::::::::::::::::::::::
'::::::::::::::::::::::::
MOVJ C00507 BC00507 VJ=50.00
MOVJ C00508 BC00508 VJ=50.00
'------------------------
'W215A
'------------------------
SFTON P0359
MOVL C00509 BC00509 V=666.7
MOVL C00510 BC00510 V=166.7 PL=0
MACRO1 MJ#(0) ARGF9
ARCON
SFTOF
SFTON P0358
MOVL C00511 BC00511 V=11.7
ARCOF
MOVL C00512 BC00512 V=333.3
SFTOF
MOVJ C00513 BC00513 VJ=50.00
MOVJ C00514 BC00514 VJ=50.00
MOVJ C00515 BC00515 VJ=50.00
MOVJ C00516 BC00516 VJ=50.00
MOVJ C00517 BC00517 VJ=50.00
MOVJ C00518 BC00518 VJ=50.00
MOVJ C00519 BC00519 VJ=50.00
MOVJ C00520 BC00520 VJ=50.00
MOVJ C00521 BC00521 VJ=50.00
'------------------------
'W31.21
'------------------------
MOVL C00522 BC00522 V=333.3
SFTON P0311
MOVL C00523 BC00523 V=166.7 PL=0
MACRO1 MJ#(0) ARGF10
ARCON
MOVL C00524 BC00524 V=10.8
ARCOF
MOVL C00525 BC00525 V=166.7
SFTOF
'------------------------
'W31.22
'------------------------
SFTON P0312
MOVL C00526 BC00526 V=666.7
MOVL C00527 BC00527 V=166.7 PL=0
ARCON
MOVL C00528 BC00528 V=10.8
ARCOF
MOVL C00529 BC00529 V=166.7
SFTOF
'------------------------
'W31.24
'------------------------
SFTON P0313
MOVL C00530 BC00530 V=666.7
MOVL C00531 BC00531 V=166.7 PL=0
ARCON
MOVL C00532 BC00532 V=10.8
ARCOF
MOVL C00533 BC00533 V=166.7
MOVL C00534 BC00534 V=166.7
MOVL C00535 BC00535 V=333.3
SFTOF
MOVL C00536 BC00536 V=333.3
MOVJ C00537 BC00537 VJ=30.00
MOVJ C00538 BC00538 VJ=30.00
MOVJ C00539 BC00539 VJ=50.00
MOVJ C00540 BC00540 VJ=50.00
COMM '::::::::::::::::::::::::
COMM '::::::::::::::::::::::::
COMM '::::::::::::::::::::::::
COMM '::::::::::::::::::::::::
COMM '::::::::::::::::::::::::
COMM '::::::::::::::::::::::::
COMM '::::::::::::::::::::::::
COMM MOVJ C00541 BC00541 VJ=50.00
COMM MOVJ C00542 BC00542 VJ=50.00
COMM '::::::::::::::::::::::::::::::::
COMM '::::::::::::::::::::::::::::::::
COMM '------------------------
COMM 'W27.19
COMM '------------------------
COMM '::::::::::::::::::::::::::::::::
COMM '::::::::::::::::::::::::::::::::
COMM MOVJ C00543 BC00543 VJ=30.00
COMM MOVL C00544 BC00544 V=666.7
COMM MOVL C00545 BC00545 V=250.0
COMM SFTON P0410
COMM MOVL C00546 BC00546 V=166.7 PL=0
COMM MACRO1 MJ#(0) ARGF24
COMM ARCON
COMM MOVL C00547 BC00547 V=7.5
COMM ARCOF
COMM MOVL C00548 BC00548 V=166.7
COMM SFTOF
COMM '------------------------
COMM 'W27.21
COMM '------------------------
COMM SFTON P0411
COMM MOVL C00549 BC00549 V=666.7
COMM MOVL C00550 BC00550 V=166.7 PL=0
COMM MACRO1 MJ#(0) ARGF24
COMM ARCON
COMM MOVL C00551 BC00551 V=7.5
COMM ARCOF
COMM MOVL C00552 BC00552 V=250.0
COMM SFTOF
COMM MOVJ C00553 BC00553 VJ=50.00
COMM MOVJ C00554 BC00554 VJ=50.00
COMM MOVJ C00555 BC00555 VJ=50.00
COMM '------------------------
COMM 'W27.22
COMM '------------------------
COMM MOVL C00556 BC00556 V=333.3
COMM MOVL C00557 BC00557 V=333.3
COMM SFTON P0412
COMM MOVL C00558 BC00558 V=166.7 PL=0
COMM MACRO1 MJ#(0) ARGF24
COMM ARCON
COMM MOVL C00559 BC00559 V=7.5
COMM ARCOF
COMM MOVL C00560 BC00560 V=200.0
COMM SFTOF
COMM '::::::::::::::::::::::::
COMM '::::::::::::::::::::::::
COMM '::::::::::::::::::::::::
COMM '::::::::::::::::::::::::
COMM '::::::::::::::::::::::::
COMM '::::::::::::::::::::::::
COMM '::::::::::::::::::::::::
COMM MOVJ C00561 BC00561 VJ=50.00
COMM MOVJ C00562 BC00562 VJ=50.00
COMM MOVJ C00563 BC00563 VJ=50.00
COMM MOVJ C00564 BC00564 VJ=50.00
MOVJ C00565 BC00565 VJ=50.00
'------------------------
'W215A
'------------------------
MOVJ C00566 BC00566 VJ=50.00
MOVJ C00567 BC00567 VJ=50.00
SFTON P0360
MOVL C00568 BC00568 V=500.0
MOVL C00569 BC00569 V=500.0
MOVL C00570 BC00570 V=166.7 PL=0
MACRO1 MJ#(0) ARGF9
ARCON
SFTOF
SFTON P0361
MOVL C00571 BC00571 V=11.7
MOVL C00572 BC00572 V=11.7
ARCOF
MOVL C00573 BC00573 V=500.0
SFTOF
MOVJ C00574 BC00574 VJ=50.00
MOVJ C00575 BC00575 VJ=50.00
MOVJ C00576 BC00576 VJ=50.00
MOVJ C00577 BC00577 VJ=80.00
MOVJ C00578 BC00578 VJ=50.00
MOVJ C00579 BC00579 VJ=50.00
MOVJ C00580 BC00580 VJ=40.00
MOVL C00581 BC00581 V=333.3
'------------------------
'W31.26
'------------------------
MOVL C00582 BC00582 V=833.3
SFTON P0314
MOVL C00583 BC00583 V=166.7 PL=0
MACRO1 MJ#(0) ARGF10
ARCON
MOVL C00584 BC00584 V=10.8
ARCOF
MOVL C00585 BC00585 V=200.0
SFTOF
'------------------------
'W31.27
'------------------------
SFTON P0315
MOVL C00586 BC00586 V=500.0
MOVL C00587 BC00587 V=166.7 PL=0
ARCON
MOVL C00588 BC00588 V=10.8
ARCOF
MOVL C00589 BC00589 V=200.0
SFTOF
MOVL C00590 BC00590 V=333.3
MOVL C00591 BC00591 V=166.7
ARCON
MOVL C00592 BC00592 V=10.8
ARCOF
SFTOF
MOVL C00593 BC00593 V=250.0
MOVL C00594 BC00594 V=250.0
MOVL C00595 BC00595 V=250.0
MOVL C00596 BC00596 V=333.3
MOVL C00597 BC00597 V=416.7
MOVJ C00598 BC00598 VJ=30.00
MOVJ C00599 BC00599 VJ=30.00
MOVJ C00600 BC00600 VJ=50.00
MOVJ C00601 BC00601 VJ=50.00
COMM '::::::::::::::::::::::::
COMM '::::::::::::::::::::::::
COMM '::::::::::::::::::::::::
COMM '::::::::::::::::::::::::
COMM '::::::::::::::::::::::::
COMM '::::::::::::::::::::::::
COMM '::::::::::::::::::::::::
COMM MOVJ C00602 BC00602 VJ=50.00
COMM MOVJ C00603 BC00603 VJ=30.00
COMM MOVJ C00604 BC00604 VJ=30.00
COMM MOVJ C00605 BC00605 VJ=40.00
COMM MOVJ C00606 BC00606 VJ=50.00
COMM '::::::::::::::::::::::::::::::::
COMM '::::::::::::::::::::::::::::::::
COMM '------------------------
COMM 'W27.24
COMM '------------------------
COMM '::::::::::::::::::::::::::::::::
COMM '::::::::::::::::::::::::::::::::
COMM SFTON P0413
COMM MOVL C00607 BC00607 V=666.7
COMM MOVL C00608 BC00608 V=500.0
COMM MOVL C00609 BC00609 V=166.7 PL=0
COMM MACRO1 MJ#(0) ARGF24
COMM ARCON
COMM MOVL C00610 BC00610 V=7.5
COMM ARCOF
COMM MOVL C00611 BC00611 V=166.7
COMM SFTOF
COMM MOVJ C00612 BC00612 VJ=30.00
COMM MOVJ C00613 BC00613 VJ=30.00
COMM MOVJ C00614 BC00614 VJ=30.00
COMM '------------------------
COMM 'W27.26
COMM '------------------------
COMM SFTON P0414
COMM MOVL C00615 BC00615 V=333.3
COMM MOVL C00616 BC00616 V=333.3
COMM MOVL C00617 BC00617 V=166.7 PL=0
COMM MACRO1 MJ#(0) ARGF24
COMM ARCON
COMM MOVL C00618 BC00618 V=6.7
COMM ARCOF
COMM MOVL C00619 BC00619 V=200.0
SFTOF
COMM '------------------------
COMM 'W27.27
COMM '------------------------
COMM SFTON P0414
COMM MOVL C00620 BC00620 V=333.3
COMM MOVL C00621 BC00621 V=166.7 PL=0
COMM MACRO1 MJ#(0) ARGF24
COMM ARCON
COMM MOVL C00622 BC00622 V=6.7
COMM ARCOF
COMM MOVL C00623 BC00623 V=200.0
SFTOF
COMM MOVL C00624 BC00624 V=500.0
COMM '::::::::::::::::::::::::
COMM '::::::::::::::::::::::::
COMM '::::::::::::::::::::::::
COMM '::::::::::::::::::::::::
COMM '::::::::::::::::::::::::
COMM '::::::::::::::::::::::::
COMM '::::::::::::::::::::::::
COMM MOVL C00625 BC00625 V=833.3
COMM MOVJ C00626 BC00626 VJ=50.00
COMM MOVJ C00627 BC00627 VJ=50.00
COMM MOVJ C00628 BC00628 VJ=50.00
MOVJ C00629 BC00629 VJ=50.00
'------------------------
'W218A
'------------------------
MOVJ C00630 BC00630 VJ=50.00
MOVJ C00631 BC00631 VJ=50.00
SFTON P0357
MOVL C00632 BC00632 V=500.0
MOVL C00633 BC00633 V=500.0
MOVL C00634 BC00634 V=166.7 PL=0
MACRO1 MJ#(0) ARGF9
ARCON
SFTOF
SFTON P0356
MOVL C00635 BC00635 V=11.7
ARCOF
MOVL C00636 BC00636 V=333.3
SFTOF
MOVJ C00637 BC00637 VJ=50.00
MOVJ C00638 BC00638 VJ=50.00
MOVJ C00639 BC00639 VJ=50.00
MOVJ C00640 BC00640 VJ=50.00
MOVJ C00641 BC00641 VJ=50.00
MOVJ C00642 BC00642 VJ=50.00
MOVL C00643 BC00643 V=500.0
'------------------------
'W31.29
'------------------------
'------------------------
'W31.31
'------------------------
MOVL C00644 BC00644 V=666.7
SFTON P0317
MOVL C00645 BC00645 V=166.7 PL=0
MACRO1 MJ#(0) ARGF10
ARCON
MOVL C00646 BC00646 V=10.8
ARCOF
MOVL C00647 BC00647 V=166.7
SFTOF
'------------------------
'W31.32
'------------------------
SFTON P0317
MOVL C00648 BC00648 V=333.3
MOVL C00649 BC00649 V=166.7 PL=0
ARCON
MOVL C00650 BC00650 V=10.8
ARCOF
MOVL C00651 BC00651 V=166.7
SFTOF
MOVL C00652 BC00652 V=416.7
SFTON P0319
MOVL C00653 BC00653 V=166.7
ARCON
MOVL C00654 BC00654 V=10.8
ARCOF
SFTOF
MOVL C00655 BC00655 V=250.0
MOVL C00656 BC00656 V=333.3
MOVL C00657 BC00657 V=416.7
MOVL C00658 BC00658 V=500.0
MOVL C00659 BC00659 V=500.0
MOVL C00660 BC00660 V=500.0
MOVJ C00661 BC00661 VJ=40.00
MOVJ C00662 BC00662 VJ=50.00
MOVJ C00663 BC00663 VJ=50.00
MOVJ C00664 BC00664 VJ=50.00
COMM '::::::::::::::::::::::::
COMM '::::::::::::::::::::::::
COMM '::::::::::::::::::::::::
COMM '::::::::::::::::::::::::
COMM '::::::::::::::::::::::::
COMM '::::::::::::::::::::::::
COMM '::::::::::::::::::::::::
COMM MOVJ C00665 BC00665 VJ=50.00
COMM MOVJ C00666 BC00666 VJ=50.00
COMM MOVJ C00667 BC00667 VJ=30.00
COMM '::::::::::::::::::::::::::::::::
COMM '::::::::::::::::::::::::::::::::
COMM '------------------------
COMM 'W27.29
COMM '------------------------
COMM '::::::::::::::::::::::::::::::::
COMM '::::::::::::::::::::::::::::::::
COMM SFTON P0416
COMM MOVL C00668 BC00668 V=666.7
COMM MOVL C00669 BC00669 V=166.7 PL=0
COMM MACRO1 MJ#(0) ARGF24
COMM ARCON
COMM MOVL C00670 BC00670 V=6.7
COMM ARCOF
COMM MOVL C00671 BC00671 V=166.7
COMM SFTOF
COMM '------------------------
COMM 'W27.31
COMM '------------------------
COMM SFTON P0417
COMM MOVL C00672 BC00672 V=666.7
COMM MOVL C00673 BC00673 V=166.7
COMM ARCON
COMM MOVL C00674 BC00674 V=7.5
COMM ARCOF
COMM MOVL C00675 BC00675 V=250.0
COMM SFTOF
COMM '------------------------
COMM 'W27.32
COMM '------------------------
COMM '::::::::::::::::::::::::
COMM '::::::::::::::::::::::::
COMM '::::::::::::::::::::::::
COMM '::::::::::::::::::::::::
COMM '::::::::::::::::::::::::
COMM '::::::::::::::::::::::::
COMM '::::::::::::::::::::::::
COMM MOVL C00676 BC00676 V=666.7
COMM MOVJ C00677 BC00677 VJ=40.00
COMM MOVJ C00678 BC00678 VJ=40.00
COMM MOVJ C00679 BC00679 VJ=40.00
COMM MOVJ C00680 BC00680 VJ=40.00
COMM MOVJ C00681 BC00681 VJ=50.00
COMM '------------------------
COMM 'W219A
COMM '------------------------
MOVJ C00682 BC00682 VJ=50.00
MOVJ C00683 BC00683 VJ=50.00
SFTON P0353
MOVL C00684 BC00684 V=666.7
MOVL C00685 BC00685 V=250.0
MOVL C00686 BC00686 V=166.7 PL=0
MACRO1 MJ#(0) ARGF9
ARCON
SFTOF
SFTON P0352
MOVL C00687 BC00687 V=11.7
ARCOF
MOVL C00688 BC00688 V=250.0
SFTOF
MOVJ C00689 BC00689 VJ=50.00
CALL JOB:FRONT_WELD_-90ST-1_5540
CALL JOB:MOVE_OUT_OF_TUNNEL
END
